(*
ExecuteSkill.Parameter[4].ID := ;
ExecuteSkill.Parameter[4].Name := '';
ExecuteSkill.Parameter[4].Value := ;
*)

(*
ExecuteSkill.Parameter[5].ID := ;
ExecuteSkill.Parameter[5].Name := '';
ExecuteSkill.Parameter[5].Value := ;
*)



ExecuteSkill();

StepDone := ExecuteSkill.Done;
END_ACTION

ACTION ST40_TransOutput_active:
//RT: 2014.11.23: Mover zum Output
StepDone := FALSE;

//Skill auswählen
ExecuteSkill.SkillID 		:= 1320;
ExecuteSkill.SkillName	 	:= 'Transport';

//Parameter setzen

ExecuteSkill.Parameter[3].ID := 3;
ExecuteSkill.Parameter[3].Name := 'Velocity';
ExecuteSkill.Parameter[3].Value := 300;



ExecuteSkill.Parameter[1].ID :=  1;
ExecuteSkill.Parameter[1].Name := 'TargetPosition X';
ExecuteSkill.Parameter[1].Value := 30 ;
ExecuteSkill.Parameter[1].StringValue := '#DP#2#XPosition';



ExecuteSkill.Parameter[2].ID := 2;
ExecuteSkill.Parameter[2].Name := 'TargetPosition Z';
ExecuteSkill.Parameter[2].Value := ZInputOutput;// ZCookieModule - ZCookieModuleCalibration - 2* Cookiethickness + toppingthickness+ Preasureheight  ;



(* ExecuteSkill.Parameter[4].ID := 4;
ExecuteSkill.Parameter[4].Name := 'Acceleration';
ExecuteSkill.Parameter[4].Value :=0 ;

*)
(*
ExecuteSkill.Parameter[5].ID := ;
ExecuteSkill.Parameter[5].Name := '';
ExecuteSkill.Parameter[5].Value := ;
*)



ExecuteSkill();

StepDone := ExecuteSkill.Done;
END_ACTION

ACTION ST43_UnblockOutput_active:
//RT: 2014.11.23: Gibt Mover Position Frei
StepDone := FALSE;

//Skill auswählen
ExecuteSkill.SkillID 		:= 1316;
ExecuteSkill.SkillName	 	:= 'Unblock';

//Parameter setzen

ExecuteSkill.Parameter[1].ID := 1;
ExecuteSkill.Parameter[1].Name := 'TaskID';
ExecuteSkill.Parameter[1].Value := Order.TaskID;


(*
ExecuteSkill.Parameter[2].ID := ;
ExecuteSkill.Parameter[2].Name := '';
ExecuteSkill.Parameter[2].Value := ;
*)

(*
ExecuteSkill.Parameter[3].ID := ;
ExecuteSkill.Parameter[3].Name := '';
ExecuteSkill.Parameter[3].Value := ;
*)

(*
ExecuteSkill.Parameter[4].ID := ;
ExecuteSkill.Parameter[4].Name := '';
ExecuteSkill.Parameter[4].Value := ;
*)

(*
ExecuteSkill.Parameter[5].ID := ;
ExecuteSkill.Parameter[5].Name := '';
ExecuteSkill.Parameter[5].Value := ;
*)



ExecuteSkill();

StepDone := ExecuteSkill.Done;
END_ACTION

ACTION ST4_Output_entry:
SectionReady := FALSE;
END_ACTION

ACTION ST3_Pump_active:
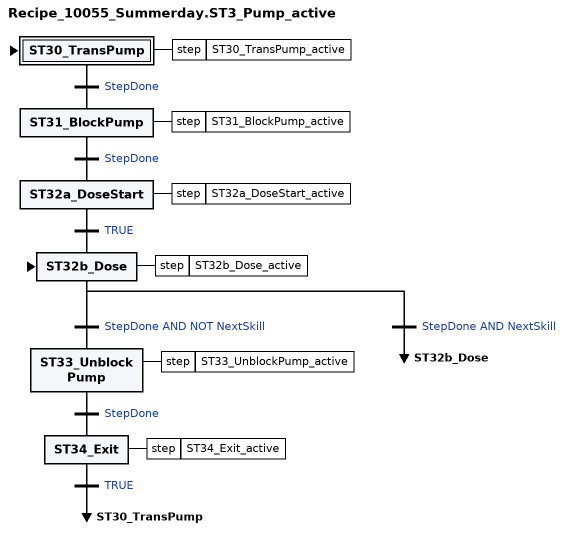
INITIAL_STEP ST30_TransPump:
    ST30_TransPump_active(N);  // step action
END_STEP
TRANSITION FROM ST30_TransPump TO ST31_BlockPump
    := StepDone;
END_TRANSITION
STEP ST31_BlockPump:
    ST31_BlockPump_active(N);  // step action
END_STEP
TRANSITION FROM ST31_BlockPump TO ST32a_DoseStart
    := StepDone;
END_TRANSITION
STEP ST32a_DoseStart:
    ST32a_DoseStart_active(N);  // step action
END_STEP
TRANSITION FROM ST32a_DoseStart TO ST32b_Dose
    := TRUE;
END_TRANSITION
STEP ST32b_Dose:
    ST32b_Dose_active(N);  // step action
END_STEP
TRANSITION FROM ST32b_Dose TO ST33_UnblockPump
    := StepDone AND NOT NextSkill;
END_TRANSITION
STEP ST33_UnblockPump:
    ST33_UnblockPump_active(N);  // step action
END_STEP
TRANSITION FROM ST33_UnblockPump TO ST34_Exit
    := StepDone;
END_TRANSITION
STEP ST34_Exit:
    ST34_Exit_active(N);  // step action
END_STEP
TRANSITION FROM ST34_Exit TO ST30_TransPump
    := TRUE;
END_TRANSITION
TRANSITION FROM ST32b_Dose TO ST32b_Dose
    := StepDone AND NextSkill;
END_TRANSITION
END_ACTION

ACTION ST41_BlockOutput_active:
//RT: 2014.11.23: Blockirt den Mover an Position
StepDone := FALSE;

//Skill auswählen
ExecuteSkill.SkillID 		:= 1315;
ExecuteSkill.SkillName	 	:= 'Block';

//Parameter setzen

ExecuteSkill.Parameter[1].ID := 1;
ExecuteSkill.Parameter[1].Name := 'TaskID';
ExecuteSkill.Parameter[1].Value := Order.TaskID;


(*
ExecuteSkill.Parameter[2].ID := ;
ExecuteSkill.Parameter[2].Name := '';
ExecuteSkill.Parameter[2].Value := ;
*)

(*
ExecuteSkill.Parameter[3].ID := ;
ExecuteSkill.Parameter[3].Name := '';
ExecuteSkill.Parameter[3].Value := ;
*)

(*
ExecuteSkill.Parameter[4].ID := ;
ExecuteSkill.Parameter[4].Name := '';
ExecuteSkill.Parameter[4].Value := ;
*)

(*
ExecuteSkill.Parameter[5].ID := ;
ExecuteSkill.Parameter[5].Name := '';
ExecuteSkill.Parameter[5].Value := ;
*)



ExecuteSkill();

StepDone := ExecuteSkill.Done;
END_ACTION

END_FUNCTION_BLOCK

// ---- POUs/Recipes/Recipe_10056_ArcturianSunrise.TcPOU
FUNCTION_BLOCK Recipe_10056_ArcturianSunrise
VAR_INPUT
	execute: BOOL;
	Order: DUT_RECIPEORDER;
END_VAR
VAR_OUTPUT
	RecipeInfo: DUT_RECIPEOFFER;
	RecipeDone: BOOL;
	InitDone: BOOL;
	Ready: BOOL;
END_VAR
VAR
	userparametersum: LREAL;
	StepDone: BOOL;
	i: INT;
	Command: ARRAY[1..5] OF DUT_RecipeCommand;
	NextSkill: BOOL;
	SectionReady: BOOL;
END_VAR

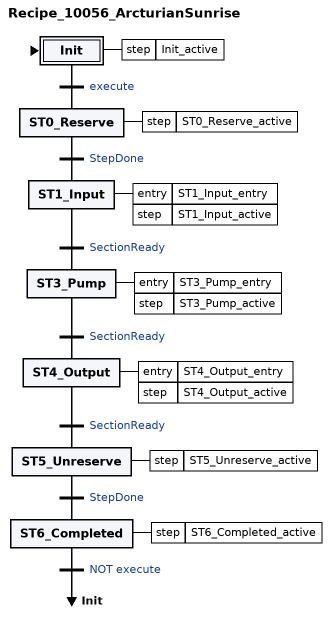
INITIAL_STEP Init:
    Init_active(N);  // step action
END_STEP
TRANSITION FROM Init TO ST0_Reserve
    := execute;
END_TRANSITION
STEP ST0_Reserve:
    ST0_Reserve_active(N);  // step action
END_STEP
TRANSITION FROM ST0_Reserve TO ST1_Input
    := StepDone;
END_TRANSITION
STEP ST1_Input:
    ST1_Input_entry(P1);  // entry action
    ST1_Input_active(N);  // step action
END_STEP
TRANSITION FROM ST1_Input TO ST3_Pump
    := SectionReady;
END_TRANSITION
STEP ST3_Pump:
    ST3_Pump_entry(P1);  // entry action
    ST3_Pump_active(N);  // step action
END_STEP
TRANSITION FROM ST3_Pump TO ST4_Output
    := SectionReady;
END_TRANSITION
STEP ST4_Output:
    ST4_Output_entry(P1);  // entry action
    ST4_Output_active(N);  // step action
END_STEP
TRANSITION FROM ST4_Output TO ST5_Unreserve
    := SectionReady;
END_TRANSITION
STEP ST5_Unreserve:
    ST5_Unreserve_active(N);  // step action
END_STEP
TRANSITION FROM ST5_Unreserve TO ST6_Completed
    := StepDone;
END_TRANSITION
STEP ST6_Completed:
    ST6_Completed_active(N);  // step action
END_STEP
TRANSITION FROM ST6_Completed TO Init
    := NOT execute;
END_TRANSITION

ACTION ST43_UnblockOutput_active:
//RT: 2014.11.23: Gibt Mover Position Frei
StepDone := FALSE;

//Skill auswählen
ExecuteSkill.SkillID 		:= 1316;
ExecuteSkill.SkillName	 	:= 'Unblock';

//Parameter setzen

ExecuteSkill.Parameter[1].ID := 1;
ExecuteSkill.Parameter[1].Name := 'TaskID';
ExecuteSkill.Parameter[1].Value := Order.TaskID;


(*
ExecuteSkill.Parameter[2].ID := ;
ExecuteSkill.Parameter[2].Name := '';
ExecuteSkill.Parameter[2].Value := ;
*)

(*
ExecuteSkill.Parameter[3].ID := ;
ExecuteSkill.Parameter[3].Name := '';
ExecuteSkill.Parameter[3].Value := ;
*)

(*
ExecuteSkill.Parameter[4].ID := ;
ExecuteSkill.Parameter[4].Name := '';
ExecuteSkill.Parameter[4].Value := ;
*)

(*
ExecuteSkill.Parameter[5].ID := ;
ExecuteSkill.Parameter[5].Name := '';
ExecuteSkill.Parameter[5].Value := ;
*)



ExecuteSkill();

StepDone := ExecuteSkill.Done;
END_ACTION

ACTION ST31_BlockPump_active:
//RT: 2014.11.23: Blockirt den Mover an Position
StepDone := FALSE;

//Skill auswählen
ExecuteSkill.SkillID 		:= 1315;
ExecuteSkill.SkillName	 	:= 'Block';

//Parameter setzen

ExecuteSkill.Parameter[1].ID := 1;
ExecuteSkill.Parameter[1].Name := 'TaskID';
ExecuteSkill.Parameter[1].Value := Order.TaskID;


(*
ExecuteSkill.Parameter[2].ID := ;
ExecuteSkill.Parameter[2].Name := '';
ExecuteSkill.Parameter[2].Value := ;
*)

(*
ExecuteSkill.Parameter[3].ID := ;
ExecuteSkill.Parameter[3].Name := '';
ExecuteSkill.Parameter[3].Value := ;
*)

(*
ExecuteSkill.Parameter[4].ID := ;
ExecuteSkill.Parameter[4].Name := '';
ExecuteSkill.Parameter[4].Value := ;
*)

(*
ExecuteSkill.Parameter[5].ID := ;
ExecuteSkill.Parameter[5].Name := '';
ExecuteSkill.Parameter[5].Value := ;
*)



ExecuteSkill();

StepDone := ExecuteSkill.Done;
END_ACTION

ACTION ST3_Pump_active:
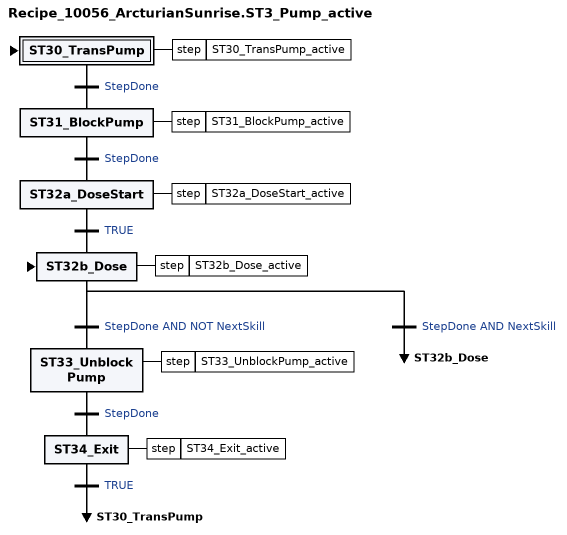
INITIAL_STEP ST30_TransPump:
    ST30_TransPump_active(N);  // step action
END_STEP
TRANSITION FROM ST30_TransPump TO ST31_BlockPump
    := StepDone;
END_TRANSITION
STEP ST31_BlockPump:
    ST31_BlockPump_active(N);  // step action
END_STEP
TRANSITION FROM ST31_BlockPump TO ST32a_DoseStart
    := StepDone;
END_TRANSITION
STEP ST32a_DoseStart:
    ST32a_DoseStart_active(N);  // step action
END_STEP
TRANSITION FROM ST32a_DoseStart TO ST32b_Dose
    := TRUE;
END_TRANSITION
STEP ST32b_Dose:
    ST32b_Dose_active(N);  // step action
END_STEP
TRANSITION FROM ST32b_Dose TO ST33_UnblockPump
    := StepDone AND NOT NextSkill;
END_TRANSITION
STEP ST33_UnblockPump:
    ST33_UnblockPump_active(N);  // step action
END_STEP
TRANSITION FROM ST33_UnblockPump TO ST34_Exit
    := StepDone;
END_TRANSITION
STEP ST34_Exit:
    ST34_Exit_active(N);  // step action
END_STEP
TRANSITION FROM ST34_Exit TO ST30_TransPump
    := TRUE;
END_TRANSITION
TRANSITION FROM ST32b_Dose TO ST32b_Dose
    := StepDone AND NextSkill;
END_TRANSITION
END_ACTION

ACTION ST44_Exit_active:
SectionReady := TRUE;
END_ACTION

ACTION ST13_UnblockInput_active:
//RT: 2014.11.23: Gibt Mover Position Frei
StepDone := FALSE;

//Skill auswählen
ExecuteSkill.SkillID 		:= 1316;
ExecuteSkill.SkillName	 	:= 'Unblock';

//Parameter setzen

ExecuteSkill.Parameter[1].ID := 1;
ExecuteSkill.Parameter[1].Name := 'TaskID';
ExecuteSkill.Parameter[1].Value := Order.TaskID;


(*
ExecuteSkill.Parameter[2].ID := ;
ExecuteSkill.Parameter[2].Name := '';
ExecuteSkill.Parameter[2].Value := ;
*)

(*
ExecuteSkill.Parameter[3].ID := ;
ExecuteSkill.Parameter[3].Name := '';
ExecuteSkill.Parameter[3].Value := ;
*)

(*
ExecuteSkill.Parameter[4].ID := ;
ExecuteSkill.Parameter[4].Name := '';
ExecuteSkill.Parameter[4].Value := ;
*)

(*
ExecuteSkill.Parameter[5].ID := ;
ExecuteSkill.Parameter[5].Name := '';
ExecuteSkill.Parameter[5].Value := ;
*)



ExecuteSkill();

StepDone := ExecuteSkill.Done;
END_ACTION

ACTION ST1_Input_active:
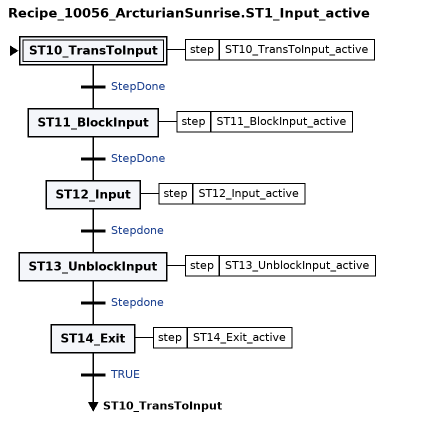
INITIAL_STEP ST10_TransToInput:
    ST10_TransToInput_active(N);  // step action
END_STEP
TRANSITION FROM ST10_TransToInput TO ST11_BlockInput
    := StepDone;
END_TRANSITION
STEP ST11_BlockInput:
    ST11_BlockInput_active(N);  // step action
END_STEP
TRANSITION FROM ST11_BlockInput TO ST12_Input
    := StepDone;
END_TRANSITION
STEP ST12_Input:
    ST12_Input_active(N);  // step action
END_STEP
TRANSITION FROM ST12_Input TO ST13_UnblockInput
    := Stepdone;
END_TRANSITION
STEP ST13_UnblockInput:
    ST13_UnblockInput_active(N);  // step action
END_STEP
TRANSITION FROM ST13_UnblockInput TO ST14_Exit
    := Stepdone;
END_TRANSITION
STEP ST14_Exit:
    ST14_Exit_active(N);  // step action
END_STEP
TRANSITION FROM ST14_Exit TO ST10_TransToInput
    := TRUE;
END_TRANSITION
END_ACTION

ACTION ST6_Completed_active:
//RT: 2014.11.23: Warte auf Execute = False
RecipeDone := TRUE;
StepDone := FALSE;
END_ACTION

ACTION ST32a_DoseStart_active:
//RT: 2014.11.23: Summe aller zutaten zum Normiren

userparametersum := 0;
FOR i := 1 TO UserParameterCnt DO
	IF NOT (order.UserParameter[i].Value = 0) THEN
		userparametersum := userparametersum + order.UserParameter[i].Value;
	
	END_IF
END_FOR
IF userparametersum = 0 THEN
userparametersum := -1;
END_IF

//RT: 2014.11.23: Start wert des Arrays setzen
i := 1;
NextSkill := TRUE ;
END_ACTION

ACTION ST11_BlockInput_active:
//RT: 2014.11.23: Blockirt den Mover an Position
StepDone := FALSE;

//Skill auswählen
ExecuteSkill.SkillID 		:= 1315;
ExecuteSkill.SkillName	 	:= 'Block';

//Parameter setzen

ExecuteSkill.Parameter[1].ID := 1;
ExecuteSkill.Parameter[1].Name := 'TaskID';
ExecuteSkill.Parameter[1].Value := Order.TaskID;


(*
ExecuteSkill.Parameter[2].ID := ;
ExecuteSkill.Parameter[2].Name := '';
ExecuteSkill.Parameter[2].Value := ;
*)

(*
ExecuteSkill.Parameter[3].ID := ;
ExecuteSkill.Parameter[3].Name := '';
ExecuteSkill.Parameter[3].Value := ;
*)

(*
ExecuteSkill.Parameter[4].ID := ;
ExecuteSkill.Parameter[4].Name := '';
ExecuteSkill.Parameter[4].Value := ;
*)

(*
ExecuteSkill.Parameter[5].ID := ;
ExecuteSkill.Parameter[5].Name := '';
ExecuteSkill.Parameter[5].Value := ;
*)



ExecuteSkill();

StepDone := ExecuteSkill.Done;
END_ACTION

ACTION ST5_Unreserve_active:
//RT: 2014.11.23: Mover Freigeben
StepDone := FALSE;

//Skill auswählen
ExecuteSkill.SkillID 		:= 1311;
ExecuteSkill.SkillName	 	:= 'Unreserve';

//Parameter setzen

ExecuteSkill.Parameter[1].ID := 1;
ExecuteSkill.Parameter[1].Name := 'TaskID';
ExecuteSkill.Parameter[1].Value := Order.TaskID;


(*
ExecuteSkill.Parameter[2].ID := ;
ExecuteSkill.Parameter[2].Name := '';
ExecuteSkill.Parameter[2].Val ue := ;
*)

(*
ExecuteSkill.Parameter[3].ID := ;
ExecuteSkill.Parameter[3].Name := '';
ExecuteSkill.Parameter[3].Value := ;
*)

(*
ExecuteSkill.Parameter[4].ID := ;
ExecuteSkill.Parameter[4].Name := '';
ExecuteSkill.Parameter[4].Value := ;
*)

(*
ExecuteSkill.Parameter[5].ID := ;
ExecuteSkill.Parameter[5].Name := '';
ExecuteSkill.Parameter[5].Value := ;
*)



ExecuteSkill();

StepDone := ExecuteSkill.Done;
END_ACTION

ACTION ST14_Exit_active:
SectionReady := TRUE;
END_ACTION

ACTION ST1_Reserve0_active:
//RT: 2014.11.23: Reservire einen Mover

StepDone := FALSE;
RecipeDone := FALSE;
//Skill auswählen
ExecuteSkill.SkillID 		:= 1310;
ExecuteSkill.SkillName	 	:= 'Reserve';

//Parameter setzen

ExecuteSkill.Parameter[1].ID := 1;
ExecuteSkill.Parameter[1].Name := 'TaskID';
ExecuteSkill.Parameter[1].Value := Order.TaskID;

(*
ExecuteSkill.Parameter[2].ID := ;
ExecuteSkill.Parameter[2].Name := '';
ExecuteSkill.Parameter[2].Value := ;
*)

(*
ExecuteSkill.Parameter[3].ID := ;
ExecuteSkill.Parameter[3].Name := '';
ExecuteSkill.Parameter[3].Value := ;
*)

(*
ExecuteSkill.Parameter[4].ID := ;
ExecuteSkill.Parameter[4].Name := '';
ExecuteSkill.Parameter[4].Value := ;
*)

(*
ExecuteSkill.Parameter[5].ID := ;
ExecuteSkill.Parameter[5].Name := '';
ExecuteSkill.Parameter[5].Value := ;
*)

ExecuteSkill();

StepDone := ExecuteSkill.Done;
END_ACTION

ACTION ST32b_Dose_active:
//RT: 2014.11.23: Die Dosir Skills anlegen
StepDone := FALSE;

//Skill auswählen
ExecuteSkill.SkillID 		:= Command[i].SkillID;
ExecuteSkill.SkillName	 	:= Command[i].SkillName;
//Parameter setzen

ExecuteSkill.Parameter[0].ID := 1;
ExecuteSkill.Parameter[0].Name := 'Quantity';
//order.userParameter[0] = amount
ExecuteSkill.Parameter[0].Value := order.UserParameter[0].Value * order.UserParameter[i].Value / userparametersum ;//Summe aller Zutatenmengen;

(*
ExecuteSkill.Parameter[2].ID := ;
ExecuteSkill.Parameter[2].Name := '';
ExecuteSkill.Parameter[2].Value := ;
*)

(*
ExecuteSkill.Parameter[3].ID := ;
ExecuteSkill.Parameter[3].Name := '';
ExecuteSkill.Parameter[3].Value := ;
*)

(*
ExecuteSkill.Parameter[4].ID := ;
ExecuteSkill.Parameter[4].Name := '';
ExecuteSkill.Parameter[4].Value := ;
*)

(*
ExecuteSkill.Parameter[5].ID := ;
ExecuteSkill.Parameter[5].Name := '';
ExecuteSkill.Parameter[5].Value := ;
*)


ExecuteSkill();

StepDone := ExecuteSkill.Done;

i := i + 1 ;

IF i = 6 THEN
	NextSkill := FALSE;
ELSIF Command[i].SkillID = 0 THEN
	NextSkill := FALSE;
ELSE
	NextSkill := TRUE;
END_IF
END_ACTION

ACTION ST3_Pump_entry:
SectionReady := FALSE;
END_ACTION

ACTION Init_active:
//RT: 2014.11.23: Vorbereiten der daten und der HMI
RecipeDone := FALSE;

// Initialisation of Recipe Parameters an name etc
RecipeInfo.Name := 'Blue Sunrise';
RecipeInfo.Description := 'Contrastful arrangement of sweet syrup and sour juice';
RecipeInfo.Dummy := FALSE;
RecipeInfo.RecipeID := 10056; 	// 
Initdone := TRUE;

//RT: 2014.11.23: wenn weniger als 5 alle lehren skills SkillID := 0
Command[1].SkillID := 1112;
Command[1].SkillName := 'Lemon Juice';
Command[1].Quantity := 30;

Command[2].SkillID := 1118;
Command[2].SkillName := 'Strawberry Syrup';
Command[2].Quantity := 8;

Command[3].SkillID := 1114;
Command[3].SkillName := 'Pineapple Juice';
Command[3].Quantity := 54;

Command[4].SkillID := 1111;
Command[4].SkillName := 'Blue Curacao';
Command[4].Quantity := 8;

Command[5].SkillID := 0;
Command[5].SkillName := 'Nothing';
Command[5].Quantity := 0;








//Parameter 0:

	RecipeInfo.UserParameter[0].Dummy 		:= FALSE;
	RecipeInfo.UserParameter[0].Default		:= 200;
	RecipeInfo.UserParameter[0].Description	:= 'Gives the total fluid amount in the glass';
	RecipeInfo.UserParameter[0].MaxValue	:= 200;
	RecipeInfo.UserParameter[0].MinValue	:= 10;
	RecipeInfo.UserParameter[0].Name		:= 'Total Liquid Amount';
	RecipeInfo.UserParameter[0].Unit		:= 'ml';
	
//Parameter 1-5:
FOR i := 1 TO 5 DO
	IF Command[i].SkillID = 0 THEN
		RecipeInfo.UserParameter[i].Dummy 		:= TRUE;
	ELSE
		RecipeInfo.UserParameter[i].Dummy 		:= FALSE;
		RecipeInfo.UserParameter[i].Default		:= Command[i].Quantity;
		RecipeInfo.UserParameter[i].Description	:= Command[i].SkillName;
		RecipeInfo.UserParameter[i].MaxValue	:= 100;
		RecipeInfo.UserParameter[i].MinValue	:= 1;
		RecipeInfo.UserParameter[i].Name		:= Command[i].SkillName;
		RecipeInfo.UserParameter[i].Unit		:= 'ml';	
	END_IF
END_FOR
END_ACTION

ACTION ST32b_Dose_exit:

END_ACTION

ACTION ST40_TransOutput_active:
//RT: 2014.11.23: Mover zum Output
StepDone := FALSE;

//Skill auswählen
ExecuteSkill.SkillID 		:= 1320;
ExecuteSkill.SkillName	 	:= 'Transport';

//Parameter setzen

ExecuteSkill.Parameter[3].ID := 3;
ExecuteSkill.Parameter[3].Name := 'Velocity';
ExecuteSkill.Parameter[3].Value := 300;



ExecuteSkill.Parameter[1].ID :=  1;
ExecuteSkill.Parameter[1].Name := 'TargetPosition X';
ExecuteSkill.Parameter[1].Value := 30 ;
ExecuteSkill.Parameter[1].StringValue := '#DP#2#XPosition';



ExecuteSkill.Parameter[2].ID := 2;
ExecuteSkill.Parameter[2].Name := 'TargetPosition Z';
ExecuteSkill.Parameter[2].Value := 100;// ZCookieModule - ZCookieModuleCalibration - 2* Cookiethickness + toppingthickness+ Preasureheight  ;



(* ExecuteSkill.Parameter[4].ID := 4;
ExecuteSkill.Parameter[4].Name := 'Acceleration';
ExecuteSkill.Parameter[4].Value :=0 ;

*)
(*
ExecuteSkill.Parameter[5].ID := ;
ExecuteSkill.Parameter[5].Name := '';
ExecuteSkill.Parameter[5].Value := ;
*)



ExecuteSkill();

StepDone := ExecuteSkill.Done;
END_ACTION

ACTION ST33_UnblockPump_active:
//RT: 2014.11.23: Gibt Mover Position Frei
StepDone := FALSE;

//Skill auswählen
ExecuteSkill.SkillID 		:= 1316;
ExecuteSkill.SkillName	 	:= 'Unblock';

//Parameter setzen

ExecuteSkill.Parameter[1].ID := 1;
ExecuteSkill.Parameter[1].Name := 'TaskID';
ExecuteSkill.Parameter[1].Value := Order.TaskID;


(*
ExecuteSkill.Parameter[2].ID := ;
ExecuteSkill.Parameter[2].Name := '';
ExecuteSkill.Parameter[2].Value := ;
*)

(*
ExecuteSkill.Parameter[3].ID := ;
ExecuteSkill.Parameter[3].Name := '';
ExecuteSkill.Parameter[3].Value := ;
*)

(*
ExecuteSkill.Parameter[4].ID := ;
ExecuteSkill.Parameter[4].Name := '';
ExecuteSkill.Parameter[4].Value := ;
*)

(*
ExecuteSkill.Parameter[5].ID := ;
ExecuteSkill.Parameter[5].Name := '';
ExecuteSkill.Parameter[5].Value := ;
*)



ExecuteSkill();

StepDone := ExecuteSkill.Done;
END_ACTION

ACTION ST0_Reserve_active:
//RT: 2014.11.23: Reservire einen Mover

StepDone := FALSE;
RecipeDone := FALSE;
//Skill auswählen
ExecuteSkill.SkillID 		:= 1310;
ExecuteSkill.SkillName	 	:= 'Reserve';

//Parameter setzen

ExecuteSkill.Parameter[1].ID := 1;
ExecuteSkill.Parameter[1].Name := 'TaskID';
ExecuteSkill.Parameter[1].Value := Order.TaskID;

(*
ExecuteSkill.Parameter[2].ID := ;
ExecuteSkill.Parameter[2].Name := '';
ExecuteSkill.Parameter[2].Value := ;
*)

(*
ExecuteSkill.Parameter[3].ID := ;
ExecuteSkill.Parameter[3].Name := '';
ExecuteSkill.Parameter[3].Value := ;
*)

(*
ExecuteSkill.Parameter[4].ID := ;
ExecuteSkill.Parameter[4].Name := '';
ExecuteSkill.Parameter[4].Value := ;
*)

(*
ExecuteSkill.Parameter[5].ID := ;
ExecuteSkill.Parameter[5].Name := '';
ExecuteSkill.Parameter[5].Value := ;
*)

ExecuteSkill();

StepDone := ExecuteSkill.Done;
END_ACTION

ACTION ST42_CocktailOutput_active:
//RT: 2014.11.23: Ausgeben des Produktes
StepDone := FALSE;

//Skill auswählen
ExecuteSkill.SkillID 		:= 1403;
ExecuteSkill.SkillName	 	:= 'Output';

//Parameter setzen

ExecuteSkill.Parameter[1].ID := 1;
ExecuteSkill.Parameter[1].Name := 'TaskID';
ExecuteSkill.Parameter[1].Value := Order.TaskID;


(*
ExecuteSkill.Parameter[2].ID := ;
ExecuteSkill.Parameter[2].Name := '';
ExecuteSkill.Parameter[2].Value := ;
*)

(*
ExecuteSkill.Parameter[3].ID := ;
ExecuteSkill.Parameter[3].Name := '';
ExecuteSkill.Parameter[3].Value := ;
*)

(*
ExecuteSkill.Parameter[4].ID := ;
ExecuteSkill.Parameter[4].Name := '';
ExecuteSkill.Parameter[4].Value := ;
*)

(*
ExecuteSkill.Parameter[5].ID := ;
ExecuteSkill.Parameter[5].Name := '';
ExecuteSkill.Parameter[5].Value := ;
*)



ExecuteSkill();

StepDone := ExecuteSkill.Done;
END_ACTION

ACTION ST4_Output_entry:
SectionReady := FALSE;
END_ACTION

ACTION ST4_Output_active:
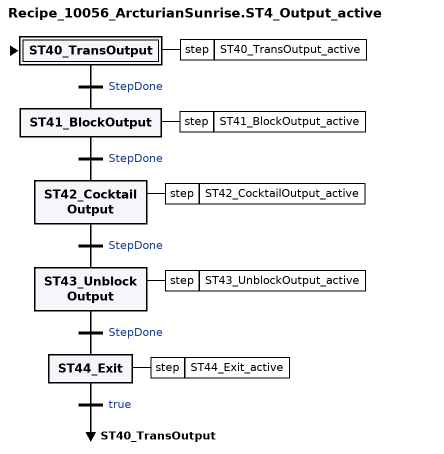
INITIAL_STEP ST40_TransOutput:
    ST40_TransOutput_active(N);  // step action
END_STEP
TRANSITION FROM ST40_TransOutput TO ST41_BlockOutput
    := StepDone;
END_TRANSITION
STEP ST41_BlockOutput:
    ST41_BlockOutput_active(N);  // step action
END_STEP
TRANSITION FROM ST41_BlockOutput TO ST42_CocktailOutput
    := StepDone;
END_TRANSITION
STEP ST42_CocktailOutput:
    ST42_CocktailOutput_active(N);  // step action
END_STEP
TRANSITION FROM ST42_CocktailOutput TO ST43_UnblockOutput
    := StepDone;
END_TRANSITION
STEP ST43_UnblockOutput:
    ST43_UnblockOutput_active(N);  // step action
END_STEP
TRANSITION FROM ST43_UnblockOutput TO ST44_Exit
    := StepDone;
END_TRANSITION
STEP ST44_Exit:
    ST44_Exit_active(N);  // step action
END_STEP
TRANSITION FROM ST44_Exit TO ST40_TransOutput
    := true;
END_TRANSITION
END_ACTION

ACTION ST30_TransPump_active:
//RT: 2014.11.23: Mover zum Pump
StepDone := FALSE;

//Skill auswählen
ExecuteSkill.SkillID 		:= 1320;
ExecuteSkill.SkillName	 	:= 'Transport';

//Parameter setzen

ExecuteSkill.Parameter[3].ID := 3;
ExecuteSkill.Parameter[3].Name := 'Velocity';
ExecuteSkill.Parameter[3].Value := 1000;



ExecuteSkill.Parameter[1].ID :=  1;
ExecuteSkill.Parameter[1].Name := 'TargetPosition X';
ExecuteSkill.Parameter[1].Value := 30 ;
ExecuteSkill.Parameter[1].StringValue := '#DP#2#XPosition';



ExecuteSkill.Parameter[2].ID := 2;
ExecuteSkill.Parameter[2].Name := 'TargetPosition Z';
ExecuteSkill.Parameter[2].Value := 25;// ZCookieModule - ZCookieModuleCalibration - 2* Cookiethickness + toppingthickness+ Preasureheight  ;



(*
ExecuteSkill.Parameter[4].ID := 4;
ExecuteSkill.Parameter[4].Name := 'Acceleration';
ExecuteSkill.Parameter[4].Value := 0 ;
*)

(*
ExecuteSkill.Parameter[5].ID := ;
ExecuteSkill.Parameter[5].Name := '';
ExecuteSkill.Parameter[5].Value := ;
*)



ExecuteSkill();

StepDone := ExecuteSkill.Done;
END_ACTION

ACTION ST10_TransToInput_active:
//RT: 2014.11.23: Mover zum Input

StepDone := FALSE;

//Skill auswählen
ExecuteSkill.SkillID 		:= 1320;
ExecuteSkill.SkillName	 	:= 'Transport';

//Parameter setzen

ExecuteSkill.Parameter[3].ID := 3;
ExecuteSkill.Parameter[3].Name := 'Velocity';
ExecuteSkill.Parameter[3].Value := 1000;



ExecuteSkill.Parameter[1].ID :=  1;
ExecuteSkill.Parameter[1].Name := 'TargetPosition X';
ExecuteSkill.Parameter[1].Value := 30 ;
ExecuteSkill.Parameter[1].StringValue := '#DP#2#XPosition';



ExecuteSkill.Parameter[2].ID := 2;
ExecuteSkill.Parameter[2].Name := 'TargetPosition Z';
ExecuteSkill.Parameter[2].Value := 100;// ZCookieModule - ZCookieModuleCalibration - 2* Cookiethickness + toppingthickness+ Preasureheight  ;



(*
ExecuteSkill.Parameter[4].ID := 4;
ExecuteSkill.Parameter[4].Name := 'Acceleration';
ExecuteSkill.Parameter[4].Value := 0 ;
*)

(*
ExecuteSkill.Parameter[5].ID := ;
ExecuteSkill.Parameter[5].Name := '';
ExecuteSkill.Parameter[5].Value := ;
*)



ExecuteSkill();

StepDone := ExecuteSkill.Done;
END_ACTION

ACTION ST12_Input_active:
//RT: 2014.11.23: Input Modul auslösen
StepDone := FALSE;

//Skill auswählen
ExecuteSkill.SkillID 		:= 1402;
ExecuteSkill.SkillName	 	:= 'Input';

//Parameter setzen

ExecuteSkill.Parameter[1].ID := 1;
ExecuteSkill.Parameter[1].Name := 'TaskID';
ExecuteSkill.Parameter[1].Value := Order.TaskID;


(*
ExecuteSkill.Parameter[2].ID := ;
ExecuteSkill.Parameter[2].Name := '';
ExecuteSkill.Parameter[2].Value := ;
*)

(*
ExecuteSkill.Parameter[3].ID := ;
ExecuteSkill.Parameter[3].Name := '';
ExecuteSkill.Parameter[3].Value := ;
*)

(*
ExecuteSkill.Parameter[4].ID := ;
ExecuteSkill.Parameter[4].Name := '';
ExecuteSkill.Parameter[4].Value := ;
*)

(*
ExecuteSkill.Parameter[5].ID := ;
ExecuteSkill.Parameter[5].Name := '';
ExecuteSkill.Parameter[5].Value := ;
*)



ExecuteSkill();

StepDone := ExecuteSkill.Done;
END_ACTION

ACTION ST41_BlockOutput_active:
//RT: 2014.11.23: Blockirt den Mover an Position
StepDone := FALSE;

//Skill auswählen
ExecuteSkill.SkillID 		:= 1315;
ExecuteSkill.SkillName	 	:= 'Block';

//Parameter setzen

ExecuteSkill.Parameter[1].ID := 1;
ExecuteSkill.Parameter[1].Name := 'TaskID';
ExecuteSkill.Parameter[1].Value := Order.TaskID;


(*
ExecuteSkill.Parameter[2].ID := ;
ExecuteSkill.Parameter[2].Name := '';
ExecuteSkill.Parameter[2].Value := ;
*)

(*
ExecuteSkill.Parameter[3].ID := ;
ExecuteSkill.Parameter[3].Name := '';
ExecuteSkill.Parameter[3].Value := ;
*)

(*
ExecuteSkill.Parameter[4].ID := ;
ExecuteSkill.Parameter[4].Name := '';
ExecuteSkill.Parameter[4].Value := ;
*)

(*
ExecuteSkill.Parameter[5].ID := ;
ExecuteSkill.Parameter[5].Name := '';
ExecuteSkill.Parameter[5].Value := ;
*)



ExecuteSkill();

StepDone := ExecuteSkill.Done;
END_ACTION

ACTION ST1_Input_entry:
SectionReady := FALSE;
END_ACTION

ACTION ST34_Exit_active:
SectionReady := TRUE;
END_ACTION

END_FUNCTION_BLOCK

// ---- POUs/Recipes/Recipe_10057_GreenFive.TcPOU
FUNCTION_BLOCK Recipe_10057_GreenFive
VAR_INPUT
	execute: BOOL;
	Order: DUT_RECIPEORDER;
END_VAR
VAR_OUTPUT
	RecipeInfo: DUT_RECIPEOFFER;
	RecipeDone: BOOL;
	InitDone: BOOL;
	Ready: BOOL;
END_VAR
VAR
	userparametersum: LREAL;
	StepDone: BOOL;
	i: INT;
	Command: ARRAY[1..5] OF DUT_RecipeCommand;
	NextSkill: BOOL;
	SectionReady: BOOL;
END_VAR

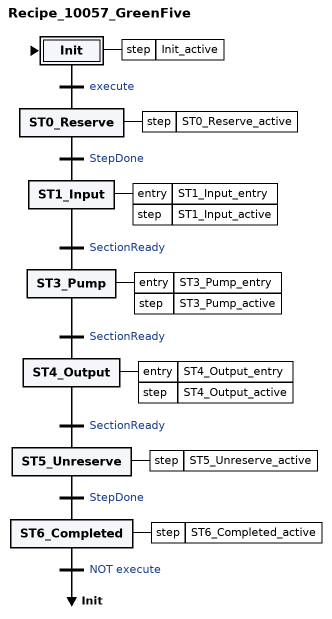
INITIAL_STEP Init:
    Init_active(N);  // step action
END_STEP
TRANSITION FROM Init TO ST0_Reserve
    := execute;
END_TRANSITION
STEP ST0_Reserve:
    ST0_Reserve_active(N);  // step action
END_STEP
TRANSITION FROM ST0_Reserve TO ST1_Input
    := StepDone;
END_TRANSITION
STEP ST1_Input:
    ST1_Input_entry(P1);  // entry action
    ST1_Input_active(N);  // step action
END_STEP
TRANSITION FROM ST1_Input TO ST3_Pump
    := SectionReady;
END_TRANSITION
STEP ST3_Pump:
    ST3_Pump_entry(P1);  // entry action
    ST3_Pump_active(N);  // step action
END_STEP
TRANSITION FROM ST3_Pump TO ST4_Output
    := SectionReady;
END_TRANSITION
STEP ST4_Output:
    ST4_Output_entry(P1);  // entry action
    ST4_Output_active(N);  // step action
END_STEP
TRANSITION FROM ST4_Output TO ST5_Unreserve
    := SectionReady;
END_TRANSITION
STEP ST5_Unreserve:
    ST5_Unreserve_active(N);  // step action
END_STEP
TRANSITION FROM ST5_Unreserve TO ST6_Completed
    := StepDone;
END_TRANSITION
STEP ST6_Completed:
    ST6_Completed_active(N);  // step action
END_STEP
TRANSITION FROM ST6_Completed TO Init
    := NOT execute;
END_TRANSITION

ACTION ST6_Completed_active:
//RT: 2014.11.23: Warte auf Execute = False
RecipeDone := TRUE;
StepDone := FALSE;
END_ACTION

ACTION ST1_Input_entry:
SectionReady := FALSE;
END_ACTION

ACTION ST3_Pump_entry:
SectionReady := FALSE;
END_ACTION

ACTION ST32b_Dose_active:
//RT: 2014.11.23: Die Dosir Skills anlegen
StepDone := FALSE;

//Skill auswählen
ExecuteSkill.SkillID 		:= Command[i].SkillID;
ExecuteSkill.SkillName	 	:= Command[i].SkillName;
//Parameter setzen

ExecuteSkill.Parameter[0].ID := 1;
ExecuteSkill.Parameter[0].Name := 'Quantity';
//order.userParameter[0] = amount
ExecuteSkill.Parameter[0].Value := order.UserParameter[0].Value * order.UserParameter[i].Value / userparametersum ;//Summe aller Zutatenmengen;

(*
ExecuteSkill.Parameter[2].ID := ;
ExecuteSkill.Parameter[2].Name := '';
ExecuteSkill.Parameter[2].Value := ;
*)

(*
ExecuteSkill.Parameter[3].ID := ;
ExecuteSkill.Parameter[3].Name := '';
ExecuteSkill.Parameter[3].Value := ;
*)

(*
ExecuteSkill.Parameter[4].ID := ;
ExecuteSkill.Parameter[4].Name := '';
ExecuteSkill.Parameter[4].Value := ;
*)

(*
ExecuteSkill.Parameter[5].ID := ;
ExecuteSkill.Parameter[5].Name := '';
ExecuteSkill.Parameter[5].Value := ;
*)


ExecuteSkill();

StepDone := ExecuteSkill.Done;

i := i + 1 ;

IF i = 6 THEN
	NextSkill := FALSE;
ELSIF Command[i].SkillID = 0 THEN
	NextSkill := FALSE;
ELSE
	NextSkill := TRUE;
END_IF
END_ACTION

ACTION ST32a_DoseStart_active:
//RT: 2014.11.23: Summe aller zutaten zum Normiren

userparametersum := 0;
FOR i := 1 TO UserParameterCnt DO
	IF NOT (order.UserParameter[i].Value = 0) THEN
		userparametersum := userparametersum + order.UserParameter[i].Value;
	
	END_IF
END_FOR
IF userparametersum = 0 THEN
userparametersum := -1;
END_IF

//RT: 2014.11.23: Start wert des Arrays setzen
i := 1;
NextSkill := TRUE ;
END_ACTION

ACTION ST12_Input_active:
//RT: 2014.11.23: Input Modul auslösen
StepDone := FALSE;

//Skill auswählen
ExecuteSkill.SkillID 		:= 1402;
ExecuteSkill.SkillName	 	:= 'Input';

//Parameter setzen

ExecuteSkill.Parameter[1].ID := 1;
ExecuteSkill.Parameter[1].Name := 'TaskID';
ExecuteSkill.Parameter[1].Value := Order.TaskID;


(*
ExecuteSkill.Parameter[2].ID := ;
ExecuteSkill.Parameter[2].Name := '';
ExecuteSkill.Parameter[2].Value := ;
*)

(*
ExecuteSkill.Parameter[3].ID := ;
ExecuteSkill.Parameter[3].Name := '';
ExecuteSkill.Parameter[3].Value := ;
*)

(*
ExecuteSkill.Parameter[4].ID := ;
ExecuteSkill.Parameter[4].Name := '';
ExecuteSkill.Parameter[4].Value := ;
*)

(*
ExecuteSkill.Parameter[5].ID := ;
ExecuteSkill.Parameter[5].Name := '';
ExecuteSkill.Parameter[5].Value := ;
*)



ExecuteSkill();

StepDone := ExecuteSkill.Done;
END_ACTION

ACTION ST3_Pump_active:
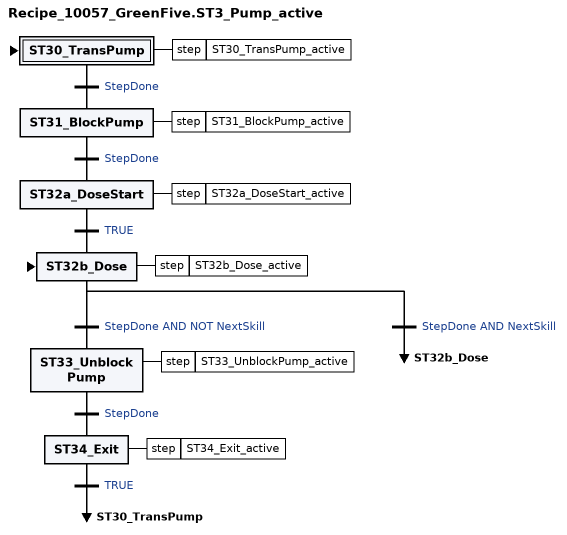
INITIAL_STEP ST30_TransPump:
    ST30_TransPump_active(N);  // step action
END_STEP
TRANSITION FROM ST30_TransPump TO ST31_BlockPump
    := StepDone;
END_TRANSITION
STEP ST31_BlockPump:
    ST31_BlockPump_active(N);  // step action
END_STEP
TRANSITION FROM ST31_BlockPump TO ST32a_DoseStart
    := StepDone;
END_TRANSITION
STEP ST32a_DoseStart:
    ST32a_DoseStart_active(N);  // step action
END_STEP
TRANSITION FROM ST32a_DoseStart TO ST32b_Dose
    := TRUE;
END_TRANSITION
STEP ST32b_Dose:
    ST32b_Dose_active(N);  // step action
END_STEP
TRANSITION FROM ST32b_Dose TO ST33_UnblockPump
    := StepDone AND NOT NextSkill;
END_TRANSITION
STEP ST33_UnblockPump:
    ST33_UnblockPump_active(N);  // step action
END_STEP
TRANSITION FROM ST33_UnblockPump TO ST34_Exit
    := StepDone;
END_TRANSITION
STEP ST34_Exit:
    ST34_Exit_active(N);  // step action
END_STEP
TRANSITION FROM ST34_Exit TO ST30_TransPump
    := TRUE;
END_TRANSITION
TRANSITION FROM ST32b_Dose TO ST32b_Dose
    := StepDone AND NextSkill;
END_TRANSITION
END_ACTION

ACTION ST34_Exit_active:
SectionReady := TRUE;
END_ACTION

ACTION ST32b_Dose_exit:

END_ACTION

ACTION ST44_Exit_active:
SectionReady := TRUE;
END_ACTION

ACTION ST10_TransToInput_active:
//RT: 2014.11.23: Mover zum Input

StepDone := FALSE;

//Skill auswählen
ExecuteSkill.SkillID 		:= 1320;
ExecuteSkill.SkillName	 	:= 'Transport';

//Parameter setzen

ExecuteSkill.Parameter[3].ID := 3;
ExecuteSkill.Parameter[3].Name := 'Velocity';
ExecuteSkill.Parameter[3].Value := 1000;



ExecuteSkill.Parameter[1].ID :=  1;
ExecuteSkill.Parameter[1].Name := 'TargetPosition X';
ExecuteSkill.Parameter[1].Value := 30 ;
ExecuteSkill.Parameter[1].StringValue := '#DP#2#XPosition';



ExecuteSkill.Parameter[2].ID := 2;
ExecuteSkill.Parameter[2].Name := 'TargetPosition Z';
ExecuteSkill.Parameter[2].Value := 100;// ZCookieModule - ZCookieModuleCalibration - 2* Cookiethickness + toppingthickness+ Preasureheight  ;



(*
ExecuteSkill.Parameter[4].ID := 4;
ExecuteSkill.Parameter[4].Name := 'Acceleration';
ExecuteSkill.Parameter[4].Value := 0 ;
*)

(*
ExecuteSkill.Parameter[5].ID := ;
ExecuteSkill.Parameter[5].Name := '';
ExecuteSkill.Parameter[5].Value := ;
*)



ExecuteSkill();

StepDone := ExecuteSkill.Done;
END_ACTION

ACTION ST4_Output_entry:
SectionReady := FALSE;
END_ACTION

ACTION ST42_CocktailOutput_active:
//RT: 2014.11.23: Ausgeben des Produktes
StepDone := FALSE;

//Skill auswählen
ExecuteSkill.SkillID 		:= 1403;
ExecuteSkill.SkillName	 	:= 'Output';

//Parameter setzen

ExecuteSkill.Parameter[1].ID := 1;
ExecuteSkill.Parameter[1].Name := 'TaskID';
ExecuteSkill.Parameter[1].Value := Order.TaskID;


(*
ExecuteSkill.Parameter[2].ID := ;
ExecuteSkill.Parameter[2].Name := '';
ExecuteSkill.Parameter[2].Value := ;
*)

(*
ExecuteSkill.Parameter[3].ID := ;
ExecuteSkill.Parameter[3].Name := '';
ExecuteSkill.Parameter[3].Value := ;
*)

(*
ExecuteSkill.Parameter[4].ID := ;
ExecuteSkill.Parameter[4].Name := '';
ExecuteSkill.Parameter[4].Value := ;
*)

(*
ExecuteSkill.Parameter[5].ID := ;
ExecuteSkill.Parameter[5].Name := '';
ExecuteSkill.Parameter[5].Value := ;
*)



ExecuteSkill();

StepDone := ExecuteSkill.Done;
END_ACTION

ACTION ST5_Unreserve_active:
//RT: 2014.11.23: Mover Freigeben
StepDone := FALSE;

//Skill auswählen
ExecuteSkill.SkillID 		:= 1311;
ExecuteSkill.SkillName	 	:= 'Unreserve';

//Parameter setzen

ExecuteSkill.Parameter[1].ID := 1;
ExecuteSkill.Parameter[1].Name := 'TaskID';
ExecuteSkill.Parameter[1].Value := Order.TaskID;


(*
ExecuteSkill.Parameter[2].ID := ;
ExecuteSkill.Parameter[2].Name := '';
ExecuteSkill.Parameter[2].Val ue := ;
*)

(*
ExecuteSkill.Parameter[3].ID := ;
ExecuteSkill.Parameter[3].Name := '';
ExecuteSkill.Parameter[3].Value := ;
*)

(*
ExecuteSkill.Parameter[4].ID := ;
ExecuteSkill.Parameter[4].Name := '';
ExecuteSkill.Parameter[4].Value := ;
*)

(*
ExecuteSkill.Parameter[5].ID := ;
ExecuteSkill.Parameter[5].Name := '';
ExecuteSkill.Parameter[5].Value := ;
*)



ExecuteSkill();

StepDone := ExecuteSkill.Done;
END_ACTION

ACTION ST11_BlockInput_active:
//RT: 2014.11.23: Blockirt den Mover an Position
StepDone := FALSE;

//Skill auswählen
ExecuteSkill.SkillID 		:= 1315;
ExecuteSkill.SkillName	 	:= 'Block';

//Parameter setzen

ExecuteSkill.Parameter[1].ID := 1;
ExecuteSkill.Parameter[1].Name := 'TaskID';
ExecuteSkill.Parameter[1].Value := Order.TaskID;


(*
ExecuteSkill.Parameter[2].ID := ;
ExecuteSkill.Parameter[2].Name := '';
ExecuteSkill.Parameter[2].Value := ;
*)

(*
ExecuteSkill.Parameter[3].ID := ;
ExecuteSkill.Parameter[3].Name := '';
ExecuteSkill.Parameter[3].Value := ;
*)

(*
ExecuteSkill.Parameter[4].ID := ;
ExecuteSkill.Parameter[4].Name := '';
ExecuteSkill.Parameter[4].Value := ;
*)

(*
ExecuteSkill.Parameter[5].ID := ;
ExecuteSkill.Parameter[5].Name := '';
ExecuteSkill.Parameter[5].Value := ;
*)



ExecuteSkill();

StepDone := ExecuteSkill.Done;
END_ACTION

ACTION ST13_UnblockInput_active:
//RT: 2014.11.23: Gibt Mover Position Frei
StepDone := FALSE;

//Skill auswählen
ExecuteSkill.SkillID 		:= 1316;
ExecuteSkill.SkillName	 	:= 'Unblock';

//Parameter setzen

ExecuteSkill.Parameter[1].ID := 1;
ExecuteSkill.Parameter[1].Name := 'TaskID';
ExecuteSkill.Parameter[1].Value := Order.TaskID;


(*
ExecuteSkill.Parameter[2].ID := ;
ExecuteSkill.Parameter[2].Name := '';
ExecuteSkill.Parameter[2].Value := ;
*)

(*
ExecuteSkill.Parameter[3].ID := ;
ExecuteSkill.Parameter[3].Name := '';
ExecuteSkill.Parameter[3].Value := ;
*)

(*
ExecuteSkill.Parameter[4].ID := ;
ExecuteSkill.Parameter[4].Name := '';
ExecuteSkill.Parameter[4].Value := ;
*)

(*
ExecuteSkill.Parameter[5].ID := ;
ExecuteSkill.Parameter[5].Name := '';
ExecuteSkill.Parameter[5].Value := ;
*)



ExecuteSkill();

StepDone := ExecuteSkill.Done;
END_ACTION

ACTION ST4_Output_active:
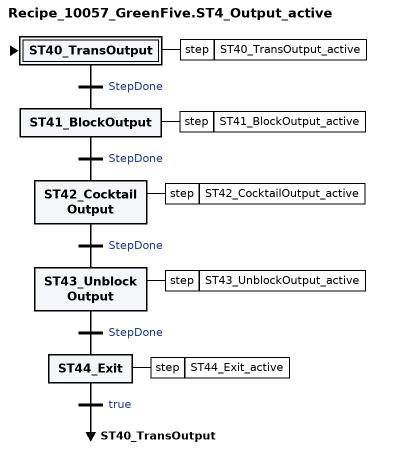
INITIAL_STEP ST40_TransOutput:
    ST40_TransOutput_active(N);  // step action
END_STEP
TRANSITION FROM ST40_TransOutput TO ST41_BlockOutput
    := StepDone;
END_TRANSITION
STEP ST41_BlockOutput:
    ST41_BlockOutput_active(N);  // step action
END_STEP
TRANSITION FROM ST41_BlockOutput TO ST42_CocktailOutput
    := StepDone;
END_TRANSITION
STEP ST42_CocktailOutput:
    ST42_CocktailOutput_active(N);  // step action
END_STEP
TRANSITION FROM ST42_CocktailOutput TO ST43_UnblockOutput
    := StepDone;
END_TRANSITION
STEP ST43_UnblockOutput:
    ST43_UnblockOutput_active(N);  // step action
END_STEP
TRANSITION FROM ST43_UnblockOutput TO ST44_Exit
    := StepDone;
END_TRANSITION
STEP ST44_Exit:
    ST44_Exit_active(N);  // step action
END_STEP
TRANSITION FROM ST44_Exit TO ST40_TransOutput
    := true;
END_TRANSITION
END_ACTION

ACTION ST0_Reserve_active:
//RT: 2014.11.23: Reservire einen Mover

StepDone := FALSE;
RecipeDone := FALSE;
//Skill auswählen
ExecuteSkill.SkillID 		:= 1310;
ExecuteSkill.SkillName	 	:= 'Reserve';

//Parameter setzen

ExecuteSkill.Parameter[1].ID := 1;
ExecuteSkill.Parameter[1].Name := 'TaskID';
ExecuteSkill.Parameter[1].Value := Order.TaskID;

(*
ExecuteSkill.Parameter[2].ID := ;
ExecuteSkill.Parameter[2].Name := '';
ExecuteSkill.Parameter[2].Value := ;
*)

(*
ExecuteSkill.Parameter[3].ID := ;
ExecuteSkill.Parameter[3].Name := '';
ExecuteSkill.Parameter[3].Value := ;
*)

(*
ExecuteSkill.Parameter[4].ID := ;
ExecuteSkill.Parameter[4].Name := '';
ExecuteSkill.Parameter[4].Value := ;
*)

(*
ExecuteSkill.Parameter[5].ID := ;
ExecuteSkill.Parameter[5].Name := '';
ExecuteSkill.Parameter[5].Value := ;
*)

ExecuteSkill();

StepDone := ExecuteSkill.Done;
END_ACTION

ACTION ST1_Reserve0_active:
//RT: 2014.11.23: Reservire einen Mover

StepDone := FALSE;
RecipeDone := FALSE;
//Skill auswählen
ExecuteSkill.SkillID 		:= 1310;
ExecuteSkill.SkillName	 	:= 'Reserve';

//Parameter setzen

ExecuteSkill.Parameter[1].ID := 1;
ExecuteSkill.Parameter[1].Name := 'TaskID';
ExecuteSkill.Parameter[1].Value := Order.TaskID;

(*
ExecuteSkill.Parameter[2].ID := ;
ExecuteSkill.Parameter[2].Name := '';
ExecuteSkill.Parameter[2].Value := ;
*)

(*
ExecuteSkill.Parameter[3].ID := ;
ExecuteSkill.Parameter[3].Name := '';
ExecuteSkill.Parameter[3].Value := ;
*)

(*
ExecuteSkill.Parameter[4].ID := ;
ExecuteSkill.Parameter[4].Name := '';
ExecuteSkill.Parameter[4].Value := ;
*)

(*
ExecuteSkill.Parameter[5].ID := ;
ExecuteSkill.Parameter[5].Name := '';
ExecuteSkill.Parameter[5].Value := ;
*)

ExecuteSkill();

StepDone := ExecuteSkill.Done;
END_ACTION

ACTION ST33_UnblockPump_active:
//RT: 2014.11.23: Gibt Mover Position Frei
StepDone := FALSE;

//Skill auswählen
ExecuteSkill.SkillID 		:= 1316;
ExecuteSkill.SkillName	 	:= 'Unblock';

//Parameter setzen

ExecuteSkill.Parameter[1].ID := 1;
ExecuteSkill.Parameter[1].Name := 'TaskID';
ExecuteSkill.Parameter[1].Value := Order.TaskID;


(*
ExecuteSkill.Parameter[2].ID := ;
ExecuteSkill.Parameter[2].Name := '';
ExecuteSkill.Parameter[2].Value := ;
*)

(*
ExecuteSkill.Parameter[3].ID := ;
ExecuteSkill.Parameter[3].Name := '';
ExecuteSkill.Parameter[3].Value := ;
*)

(*
ExecuteSkill.Parameter[4].ID := ;
ExecuteSkill.Parameter[4].Name := '';
ExecuteSkill.Parameter[4].Value := ;
*)

(*
ExecuteSkill.Parameter[5].ID := ;
ExecuteSkill.Parameter[5].Name := '';
ExecuteSkill.Parameter[5].Value := ;
*)



ExecuteSkill();

StepDone := ExecuteSkill.Done;
END_ACTION

ACTION ST43_UnblockOutput_active:
//RT: 2014.11.23: Gibt Mover Position Frei
StepDone := FALSE;

//Skill auswählen
ExecuteSkill.SkillID 		:= 1316;
ExecuteSkill.SkillName	 	:= 'Unblock';

//Parameter setzen

ExecuteSkill.Parameter[1].ID := 1;
ExecuteSkill.Parameter[1].Name := 'TaskID';
ExecuteSkill.Parameter[1].Value := Order.TaskID;


(*
ExecuteSkill.Parameter[2].ID := ;
ExecuteSkill.Parameter[2].Name := '';
ExecuteSkill.Parameter[2].Value := ;
*)

(*
ExecuteSkill.Parameter[3].ID := ;
ExecuteSkill.Parameter[3].Name := '';
ExecuteSkill.Parameter[3].Value := ;
*)

(*
ExecuteSkill.Parameter[4].ID := ;
ExecuteSkill.Parameter[4].Name := '';
ExecuteSkill.Parameter[4].Value := ;
*)

(*
ExecuteSkill.Parameter[5].ID := ;
ExecuteSkill.Parameter[5].Name := '';
ExecuteSkill.Parameter[5].Value := ;
*)



ExecuteSkill();

StepDone := ExecuteSkill.Done;
END_ACTION

ACTION ST14_Exit_active:
SectionReady := TRUE;
END_ACTION

ACTION ST41_BlockOutput_active:
//RT: 2014.11.23: Blockirt den Mover an Position
StepDone := FALSE;

//Skill auswählen
ExecuteSkill.SkillID 		:= 1315;
ExecuteSkill.SkillName	 	:= 'Block';

//Parameter setzen

ExecuteSkill.Parameter[1].ID := 1;
ExecuteSkill.Parameter[1].Name := 'TaskID';
ExecuteSkill.Parameter[1].Value := Order.TaskID;


(*
ExecuteSkill.Parameter[2].ID := ;
ExecuteSkill.Parameter[2].Name := '';
ExecuteSkill.Parameter[2].Value := ;
*)

(*
ExecuteSkill.Parameter[3].ID := ;
ExecuteSkill.Parameter[3].Name := '';
ExecuteSkill.Parameter[3].Value := ;
*)

(*
ExecuteSkill.Parameter[4].ID := ;
ExecuteSkill.Parameter[4].Name := '';
ExecuteSkill.Parameter[4].Value := ;
*)

(*
ExecuteSkill.Parameter[5].ID := ;
ExecuteSkill.Parameter[5].Name := '';
ExecuteSkill.Parameter[5].Value := ;
*)



ExecuteSkill();

StepDone := ExecuteSkill.Done;
END_ACTION

ACTION ST30_TransPump_active:
//RT: 2014.11.23: Mover zum Pump
StepDone := FALSE;

//Skill auswählen
ExecuteSkill.SkillID 		:= 1320;
ExecuteSkill.SkillName	 	:= 'Transport';

//Parameter setzen

ExecuteSkill.Parameter[3].ID := 3;
ExecuteSkill.Parameter[3].Name := 'Velocity';
ExecuteSkill.Parameter[3].Value := 1000;



ExecuteSkill.Parameter[1].ID :=  1;
ExecuteSkill.Parameter[1].Name := 'TargetPosition X';
ExecuteSkill.Parameter[1].Value := 30 ;
ExecuteSkill.Parameter[1].StringValue := '#DP#2#XPosition';



ExecuteSkill.Parameter[2].ID := 2;
ExecuteSkill.Parameter[2].Name := 'TargetPosition Z';
ExecuteSkill.Parameter[2].Value := 25;// ZCookieModule - ZCookieModuleCalibration - 2* Cookiethickness + toppingthickness+ Preasureheight  ;



(*
ExecuteSkill.Parameter[4].ID := 4;
ExecuteSkill.Parameter[4].Name := 'Acceleration';
ExecuteSkill.Parameter[4].Value := 0 ;
*)

(*
ExecuteSkill.Parameter[5].ID := ;
ExecuteSkill.Parameter[5].Name := '';
ExecuteSkill.Parameter[5].Value := ;
*)



ExecuteSkill();

StepDone := ExecuteSkill.Done;
END_ACTION

ACTION ST40_TransOutput_active:
//RT: 2014.11.23: Mover zum Output
StepDone := FALSE;

//Skill auswählen
ExecuteSkill.SkillID 		:= 1320;
ExecuteSkill.SkillName	 	:= 'Transport';

//Parameter setzen

ExecuteSkill.Parameter[3].ID := 3;
ExecuteSkill.Parameter[3].Name := 'Velocity';
ExecuteSkill.Parameter[3].Value := 300;



ExecuteSkill.Parameter[1].ID :=  1;
ExecuteSkill.Parameter[1].Name := 'TargetPosition X';
ExecuteSkill.Parameter[1].Value := 30 ;
ExecuteSkill.Parameter[1].StringValue := '#DP#2#XPosition';



ExecuteSkill.Parameter[2].ID := 2;
ExecuteSkill.Parameter[2].Name := 'TargetPosition Z';
ExecuteSkill.Parameter[2].Value := ZInputOutput;// ZCookieModule - ZCookieModuleCalibration - 2* Cookiethickness + toppingthickness+ Preasureheight  ;



(* ExecuteSkill.Parameter[4].ID := 4;
ExecuteSkill.Parameter[4].Name := 'Acceleration';
ExecuteSkill.Parameter[4].Value :=0 ;

*)
(*
ExecuteSkill.Parameter[5].ID := ;
ExecuteSkill.Parameter[5].Name := '';
ExecuteSkill.Parameter[5].Value := ;
*)



ExecuteSkill();

StepDone := ExecuteSkill.Done;
END_ACTION

ACTION Init_active:
//RT: 2014.11.23: Vorbereiten der daten und der HMI
RecipeDone := FALSE;

// Initialisation of Recipe Parameters an name etc
RecipeInfo.Name := 'Green Five';
RecipeInfo.Description := 'Remember spring feelings in autumn';
RecipeInfo.Dummy := FALSE;
RecipeInfo.RecipeID := 10057; 	// 
Initdone := TRUE;

//RT: 2014.11.23: wenn weniger als 5 alle lehren skills SkillID := 0
Command[1].SkillID := 1117;
Command[1].SkillName := 'Orange Juice';
Command[1].Quantity := 20;

Command[2].SkillID := 1112;
Command[2].SkillName := 'Lemon Juice';
Command[2].Quantity := 10;

Command[3].SkillID := 1114;
Command[3].SkillName := 'Pineapple Juice';
Command[3].Quantity := 30;

Command[4].SkillID := 1113;
Command[4].SkillName := 'Maracuja Juice';
Command[4].Quantity := 30;

Command[5].SkillID := 1119;
Command[5].SkillName := 'Blue Curacao';
Command[5].Quantity := 10;








//Parameter 0:

	RecipeInfo.UserParameter[0].Dummy 		:= FALSE;
	RecipeInfo.UserParameter[0].Default		:= 200;
	RecipeInfo.UserParameter[0].Description	:= 'Gives the total fluid amount in the glass';
	RecipeInfo.UserParameter[0].MaxValue	:= 200;
	RecipeInfo.UserParameter[0].MinValue	:= 10;
	RecipeInfo.UserParameter[0].Name		:= 'Total Liquid Amount';
	RecipeInfo.UserParameter[0].Unit		:= 'ml';
	
//Parameter 1-5:
FOR i := 1 TO 5 DO
	IF Command[i].SkillID = 0 THEN
		RecipeInfo.UserParameter[i].Dummy 		:= TRUE;
	ELSE
		RecipeInfo.UserParameter[i].Dummy 		:= FALSE;
		RecipeInfo.UserParameter[i].Default		:= Command[i].Quantity;
		RecipeInfo.UserParameter[i].Description	:= Command[i].SkillName;
		RecipeInfo.UserParameter[i].MaxValue	:= 100;
		RecipeInfo.UserParameter[i].MinValue	:= 1;
		RecipeInfo.UserParameter[i].Name		:= Command[i].SkillName;
		RecipeInfo.UserParameter[i].Unit		:= 'ml';	
	END_IF
END_FOR
END_ACTION

ACTION ST1_Input_active:
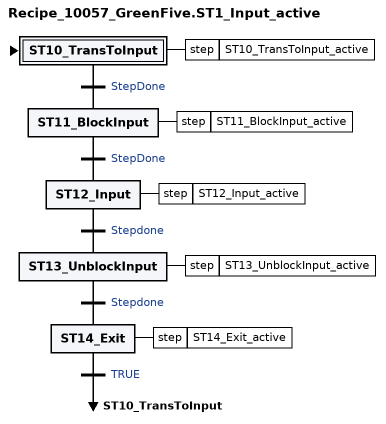
INITIAL_STEP ST10_TransToInput:
    ST10_TransToInput_active(N);  // step action
END_STEP
TRANSITION FROM ST10_TransToInput TO ST11_BlockInput
    := StepDone;
END_TRANSITION
STEP ST11_BlockInput:
    ST11_BlockInput_active(N);  // step action
END_STEP
TRANSITION FROM ST11_BlockInput TO ST12_Input
    := StepDone;
END_TRANSITION
STEP ST12_Input:
    ST12_Input_active(N);  // step action
END_STEP
TRANSITION FROM ST12_Input TO ST13_UnblockInput
    := Stepdone;
END_TRANSITION
STEP ST13_UnblockInput:
    ST13_UnblockInput_active(N);  // step action
END_STEP
TRANSITION FROM ST13_UnblockInput TO ST14_Exit
    := Stepdone;
END_TRANSITION
STEP ST14_Exit:
    ST14_Exit_active(N);  // step action
END_STEP
TRANSITION FROM ST14_Exit TO ST10_TransToInput
    := TRUE;
END_TRANSITION
END_ACTION

ACTION ST31_BlockPump_active:
//RT: 2014.11.23: Blockirt den Mover an Position
StepDone := FALSE;

//Skill auswählen
ExecuteSkill.SkillID 		:= 1315;
ExecuteSkill.SkillName	 	:= 'Block';

//Parameter setzen

ExecuteSkill.Parameter[1].ID := 1;
ExecuteSkill.Parameter[1].Name := 'TaskID';
ExecuteSkill.Parameter[1].Value := Order.TaskID;


(*
ExecuteSkill.Parameter[2].ID := ;
ExecuteSkill.Parameter[2].Name := '';
ExecuteSkill.Parameter[2].Value := ;
*)

(*
ExecuteSkill.Parameter[3].ID := ;
ExecuteSkill.Parameter[3].Name := '';
ExecuteSkill.Parameter[3].Value := ;
*)

(*
ExecuteSkill.Parameter[4].ID := ;
ExecuteSkill.Parameter[4].Name := '';
ExecuteSkill.Parameter[4].Value := ;
*)

(*
ExecuteSkill.Parameter[5].ID := ;
ExecuteSkill.Parameter[5].Name := '';
ExecuteSkill.Parameter[5].Value := ;
*)



ExecuteSkill();

StepDone := ExecuteSkill.Done;
END_ACTION

END_FUNCTION_BLOCK

// ---- POUs/FB_INIT_RECIPE.TcPOU
FUNCTION_BLOCK FB_INIT_RECIPE
VAR_INPUT
	Execute	: 	BOOL;
END_VAR
VAR_OUTPUT
	Done	: BOOL;
	Busy	: BOOL;
	Error	: BOOL;
END_VAR
VAR
	i	: INT := 10000;
	OfferCounter	: INT;
	InitOrder		: DUT_RECIPEORDER;
	fbExecuteRecipe	: FB_ExecuteRecipe;
	state: INT;
END_VAR

IF Execute THEN
	Done := FALSE;
	CASE state OF
		

		0: 
			fbExecuteRecipe.Execute := TRUE;
			InitOrder.RecipeID := i;
			state := 1;
			
		1:	
			fbExecuteRecipe(Order:= InitOrder);
			IF fbExecuteRecipe.Done THEN
				IF fbExecuteRecipe.NotAvailable THEN
				state := 50;
				ELSE
				Offer[OfferCounter]:=fbExecuteRecipe.RecipeInfo;
				OfferCounter := OfferCounter +1;
				state := 50;
				END_IF
			END_IF	
			
			
			
			
		50: IF i< 10100 THEN
				i := i+1;
				state :=0;
			ELSE
				busy 	:= FALSE;
				done 	:= TRUE;
				Execute := FALSE;
				state := 0;
			END_IF
		
		
		
		
		
		

	END_CASE
END_IF

END_FUNCTION_BLOCK

// ---- POUs/OPC/FB_ReadReset.TcPOU
FUNCTION_BLOCK FB_ReadReset
VAR_INPUT
	ReadIdentifier: STRING[80];
	NamespaceIndex: UINT;
	ConnectionHdl: DWORD;
	execute: BOOL;
END_VAR
VAR_OUTPUT
	ReadData		: BOOL;
	done: BOOL;
	busy: BOOL;
	error: BOOL;
END_VAR
VAR
		/// FBs
	fbNodeGetHandle: UA_NodeGetHandle;
	fbReadVariable: UA_Read;
	///Variables
	pReadData		: POINTER TO BOOL;
	
	VariableSize: UDINT;
	NodeHdl: DWORD;
	cbDataR: UDINT;
	state: INT := -1;
	SessionNodeID: ST_UANodeID;
	Timeout: TIME := DEFAULT_ADS_TIMEOUT;
END_VAR

IF execute THEN 
	DONE := FALSE;
	CASE state OF
		
		-1:	SessionNodeID.nNamespaceIndex    			:= Namespaceindex;
			SessionNodeID.eIdentifierType				:= 1;
			SessionNodeID.sIdentifier					:= ReadIdentifier;
			VariableSize 								:= SIZEOF (ReadData);
			pReadData									:= ADR(ReadData);
			
			
			

			busy := TRUE;
			done := FALSE;
			state:=0;

		0: fbNodeGetHandle(
			Execute:=FALSE,
			ConnectionHdl:=ConnectionHdl,
			NodeID:=SessionNodeID,
			Timeout:=Timeout,
			NodeHdl=>NodeHdl,
			Done=>,
			Busy=>busy,
			Error=>,
			ErrorID=>,);
			state:=1;
			
			
		1:fbNodeGetHandle(
			Execute:=TRUE,
			ConnectionHdl:=ConnectionHdl,
			NodeID:=SessionNodeID,
			Timeout:=Timeout,
			NodeHdl=>NodeHdl,
			Done=>,
			Busy=>busy,
			Error=>,
			ErrorID=>,);
			IF fbNodeGetHandle.Done THEN
			state := 2;
			END_IF
			IF fbNodeGetHandle.Error THEN
				state := -1;
			END_IF
		2:
			fbReadVariable(
				Execute:= FALSE, 
				ConnectionHdl:= ConnectionHdl, 
				NodeHdl:= NodeHdl, 
				stNodeAddInfo:= , 
				pVariable:= pReadData, 
				cbData:= VariableSize, 
				Timeout:= DEFAULT_ADS_TIMEOUT, 
				Done=> , 
				Busy=> , 
				Error=> , 
				ErrorID=> , 
				cbData_R=>cbDataR );
				state := 3;
				error :=FALSE;
				
		3:		fbReadVariable(
				Execute:= TRUE, 
				ConnectionHdl:= ConnectionHdl, 
				NodeHdl:= NodeHdl, 
				stNodeAddInfo:=, 
				pVariable:= pReadData, 
				cbData:= VariableSize, 
				Timeout:= DEFAULT_ADS_TIMEOUT, 
				Done=>, 
				Busy=>, 
				Error=>error, 
				ErrorID=>, 
				cbData_R=>cbDataR );
				IF fbReadVariable.Done THEN
					state		:= 2;
					execute		:= FALSE;
					done		:= TRUE;
					busy		:= FALSE;
				END_IF	
				IF fbReadVariable.Error THEN
				state := -1;
				END_IF	
		
	END_CASE
ELSE
	state := -1;
END_IF

END_FUNCTION_BLOCK

// ---- POUs/OPC/FB_WriteReset.TcPOU
FUNCTION_BLOCK FB_WriteReset
VAR_INPUT
	WriteIdentifier: STRING[80];
	NamespaceIndex: UINT;
	ConnectionHdl: DWORD;
	execute: BOOL;
	WriteData:  BOOL;
END_VAR
VAR_OUTPUT
	done: BOOL;
	busy: BOOL;
	error: BOOL;
END_VAR
VAR
	/// FBs
	fbWriteVariable: UA_Write;
	fbNodeGetHandle: UA_NodeGetHandle;
	fbNodeReleaseHandle	: UA_NodeReleaseHandle;
	/// Variables
	state: INT := -1;
	pWriteData: POINTER TO BOOL;
	VariableSize: UDINT;
	NodeHdl: DWORD;
	Timeout: TIME := DEFAULT_ADS_TIMEOUT;
	SessionNodeID: ST_UANodeID;
	Timer	: TON;
END_VAR

IF execute THEN
	Done := FALSE;
	CASE state OF
		
		-1:	SessionNodeID.nNamespaceIndex    			:= Namespaceindex;
			SessionNodeID.eIdentifierType				:= 1;
			SessionNodeID.sIdentifier					:= WriteIdentifier;
			VariableSize 								:= SIZEOF (WriteData);
			pWriteData									:= ADR(WriteData);
			
			
			done := FALSE;
			state:=0;
		
	    0: fbNodeGetHandle(
			Execute:=FALSE,
			ConnectionHdl:=ConnectionHdl,
			NodeID:=SessionNodeID,
			Timeout:=Timeout,
			NodeHdl=>NodeHdl,
			Done=>,
			Busy=>,
			Error=>,
			ErrorID=>,);
			state:=1;
			
		1:fbNodeGetHandle(
			Execute:=TRUE,
			ConnectionHdl:=ConnectionHdl,
			NodeID:=SessionNodeID,
			Timeout:=Timeout,
			NodeHdl=>NodeHdl,
			Done=>,
			Busy=>,
			Error=>,
			ErrorID=>,);
			IF fbNodeGetHandle.Done THEN
			state := 2;
			END_IF
			
		
				
		2: fbWriteVariable(
				Execute:=FALSE , 
				ConnectionHdl:=ConnectionHdl , 
				NodeHdl:=NodeHdl , 
				stNodeAddInfo:= , 
				pVariable:= pWriteData, 
				cbData:= VariableSize, 
				Timeout:=Timeout , 
				Done=> , 
				Busy=> , 
				Error=> , 
				ErrorID=> );
				
				state:=3;
				
		3: fbWriteVariable(
				Execute:=TRUE , 
				ConnectionHdl:=ConnectionHdl , 
				NodeHdl:=NodeHdl , 
				stNodeAddInfo:= , 
				pVariable:= pWriteData, 
				cbData:= VariableSize, 
				Timeout:=Timeout , 
				Done=> , 
				Busy=> , 
				Error=> , 
				ErrorID=> );
				IF fbWriteVariable.Done THEN
					state := 4;
				END_IF
				
		4: fbNodeReleaseHandle(ConnectionHdl := ConnectionHdl, Execute := FALSE, NodeHdl := NodeHdl, Timeout := Timeout);
			state := 5;
			Timer(IN := FALSE, PT := T#10S);
		5: 
			fbNodeReleaseHandle(ConnectionHdl := ConnectionHdl, Execute := TRUE, NodeHdl := NodeHdl, Timeout := Timeout);
				IF fbNodeReleaseHandle.Done OR Timer.Q THEN
					state		:= -1;
					execute		:= FALSE;
					done		:= TRUE;
					busy		:= FALSE;
				END_IF
			Timer(IN := TRUE);
			
				
	END_CASE
ELSE
	state := -1;
END_IF

END_FUNCTION_BLOCK

// ---- POUs/OPC/FB_OPCServerConnect.TcPOU
FUNCTION_BLOCK FB_OPCServerConnect
VAR_INPUT
	ServerUrl: STRING[80];
	NamespaceUri: STRING[80];
	ClientName: STRING[80];
	execute: BOOL;
END_VAR
VAR_OUTPUT
	ConnectHdl: DWORD;
	Namespaceindex: UINT;
	busy: BOOL;
	done: BOOL;
	error: BOOL;
END_VAR
VAR
	fbGetNameSpace: UA_GetNameSpaceIndex;
	SessionconnectInfo: ST_UASessionConnectInfo;
	Timeout: TIME := DEFAULT_ADS_TIMEOUT;
	state: INT := -1;
	fbConnect: UA_Connect;
END_VAR

IF execute THEN
	CASE state OF
	-1: 	SessionconnectInfo.sApplicationName			:=ClientName;
			SessionconnectInfo.eSecurityMode				:=1; 
			SessionconnectInfo.eSecurityPolicyUri		:=1;
			SessionconnectInfo.eTransportProfileUri		:=1;
			SessionconnectInfo.tConnectTimeout			:=T#4S;
			SessionconnectInfo.tSessionTimeout			:=T#3S;
			
			
			busy 	:= TRUE;
			done	:= FALSE;							
			state 	:= 0;

	0:
         fbConnect(
			Execute:= FALSE, 
			ServerUrl:=ServerUrl , 
			SessionConnectInfo:= SessionconnectInfo, 
			Timeout:= Timeout, 
			ConnectionHdl=> ConnectHdl, 
			Done=>, 
			Busy=>busy, 
			Error=>error, 
			ErrorID=>);
			
	 		state := 1;
			
	1:
         fbConnect(
			Execute:= TRUE, 
			ServerUrl:=ServerUrl , 
			SessionConnectInfo:= SessionconnectInfo, 
			Timeout:= Timeout, 
			ConnectionHdl=> ConnectHdl,  
			Done=>, 
			Busy=>busy, 
			Error=>error, 
			ErrorID=> );
			
			IF fbConnect.done THEN
			
			state := 2;
			END_IF
			
			IF fbConnect.Error THEN
				error := TRUE;
			state := 0;
			END_IF
		

			
 		
		
	2:	
		fbGetNameSpace(
			Execute:= FALSE,
			ConnectionHdl:=ConnectHdl,
			NamespaceUri:=NamespaceUri,
			Timeout:=Timeout,
			NamespaceIndex=>Namespaceindex,
			Done=>,
			Busy=>busy,
			Error=>error,
			ErrorID=>,);	
			
			state := 3;	
	3:
		fbGetNameSpace(
			Execute:= TRUE,
			ConnectionHdl:=ConnectHdl,
			NamespaceUri:=NamespaceUri,
			Timeout:=Timeout,
			NamespaceIndex=>Namespaceindex,
			Done=>,
			Busy=>busy,
			Error=>error,
			ErrorID=>,);
			IF fbGetNameSpace.done THEN
			Execute := FALSE;
			busy	:= FALSE;
			done	:= TRUE;
			state 	:= 0;
			END_IF
		END_CASE
ELSE
	done	:= FALSE;
	busy := FALSE;
	error := FALSE;
	state := -1;
END_IF

END_FUNCTION_BLOCK

// ---- POUs/OPC/FB_WriteOfferlist.TcPOU
FUNCTION_BLOCK FB_WriteOfferlist
VAR_INPUT
	WriteIdentifier: STRING[80];
	NamespaceIndex: UINT;
	ConnectionHdl: DWORD;
	execute: BOOL;
	WriteData:  ARRAY [0..OfferCnt] OF DUT_RECIPEOFFER;
END_VAR
VAR_OUTPUT
	done: BOOL;
	busy: BOOL;
	error: BOOL;
END_VAR
VAR
	/// FBs
	fbWriteVariable: UA_Write;
	fbNodeGetHandle: UA_NodeGetHandle;
	/// Variables
	state: INT := -1;
	pWriteData: POINTER TO DUT_RECIPEOFFER;
	VariableSize: UDINT;
	NodeHdl: DWORD;
	Timeout: TIME := DEFAULT_ADS_TIMEOUT;
	SessionNodeID: ST_UANodeID;
END_VAR

IF execute THEN
	CASE state OF
		
		-1:	SessionNodeID.nNamespaceIndex    			:= Namespaceindex;
			SessionNodeID.eIdentifierType				:= 1;
			SessionNodeID.sIdentifier					:= WriteIdentifier;
			VariableSize 								:= SIZEOF (WriteData);
			pWriteData								:= ADR(WriteData);
			
			
			done := FALSE;
			state:=0;
		
	    0: fbNodeGetHandle(
			Execute:=FALSE,
			ConnectionHdl:=ConnectionHdl,
			NodeID:=SessionNodeID,
			Timeout:=Timeout,
			NodeHdl=>NodeHdl,
			Done=>,
			Busy=>,
			Error=>,
			ErrorID=>,);
			state:=1;
			
		1:fbNodeGetHandle(
			Execute:=TRUE,
			ConnectionHdl:=ConnectionHdl,
			NodeID:=SessionNodeID,
			Timeout:=Timeout,
			NodeHdl=>NodeHdl,
			Done=>,
			Busy=>,
			Error=>,
			ErrorID=>,);
			IF fbNodeGetHandle.Done THEN
			state := 2;
			END_IF
			
		
				
		2: fbWriteVariable(
				Execute:=FALSE , 
				ConnectionHdl:=ConnectionHdl , 
				NodeHdl:=NodeHdl , 
				stNodeAddInfo:= , 
				pVariable:= pWriteData, 
				cbData:= VariableSize, 
				Timeout:=Timeout , 
				Done=> , 
				Busy=> , 
				Error=> , 
				ErrorID=> );
				
				state:=3;
				
		3: fbWriteVariable(
				Execute:=TRUE , 
				ConnectionHdl:=ConnectionHdl , 
				NodeHdl:=NodeHdl , 
				stNodeAddInfo:= , 
				pVariable:= pWriteData, 
				cbData:= VariableSize, 
				Timeout:=Timeout , 
				Done=> , 
				Busy=> , 
				Error=> , 
				ErrorID=> );
				IF fbWriteVariable.Done THEN
					state		:= 2;
					execute		:= FALSE;
					done		:= TRUE;
					busy		:= FALSE;
				END_IF		
	END_CASE
ELSE
	state := -1;
END_IF

END_FUNCTION_BLOCK

// ---- POUs/OPC/FB_ReadQueue.TcPOU
FUNCTION_BLOCK FB_ReadQueue
VAR_INPUT
	ReadIdentifier: STRING[80];
	NamespaceIndex: UINT;
	ConnectionHdl: DWORD;
	execute: BOOL;
END_VAR
VAR_OUTPUT
	ReadData		: DUT_RECIPEORDER;
	done: BOOL;
	busy: BOOL;
	error: BOOL;
END_VAR
VAR
		/// FBs
	fbNodeGetHandle: UA_NodeGetHandle;
	fbReadVariable: UA_Read;
	///Variables
	pReadData		: POINTER TO DUT_RECIPEORDER;
	
	VariableSize: UDINT;
	NodeHdl: DWORD;
	cbDataR: UDINT;
	state: INT := -1;
	SessionNodeID: ST_UANodeID;
	Timeout: TIME := DEFAULT_ADS_TIMEOUT;
END_VAR

IF execute THEN 
	DONE := FALSE;
	CASE state OF
		
		-1:	SessionNodeID.nNamespaceIndex    			:= Namespaceindex;
			SessionNodeID.eIdentifierType				:= 1;
			SessionNodeID.sIdentifier					:= ReadIdentifier;
			VariableSize 								:= SIZEOF (ReadData);
			pReadData									:= ADR(ReadData);
			
			
			

			busy := TRUE;
			done := FALSE;
			state:=0;

		0: fbNodeGetHandle(
			Execute:=FALSE,
			ConnectionHdl:=ConnectionHdl,
			NodeID:=SessionNodeID,
			Timeout:=Timeout,
			NodeHdl=>NodeHdl,
			Done=>,
			Busy=>busy,
			Error=>,
			ErrorID=>,);
			state:=1;
			
		1:fbNodeGetHandle(
			Execute:=TRUE,
			ConnectionHdl:=ConnectionHdl,
			NodeID:=SessionNodeID,
			Timeout:=Timeout,
			NodeHdl=>NodeHdl,
			Done=>,
			Busy=>busy,
			Error=>,
			ErrorID=>,);
			IF fbNodeGetHandle.Done THEN
			state := 2;
			END_IF
			
		2:
			fbReadVariable(
				Execute:= FALSE, 
				ConnectionHdl:= ConnectionHdl, 
				NodeHdl:= NodeHdl, 
				stNodeAddInfo:= , 
				pVariable:= pReadData, 
				cbData:= VariableSize, 
				Timeout:= DEFAULT_ADS_TIMEOUT, 
				Done=> , 
				Busy=> , 
				Error=> , 
				ErrorID=> , 
				cbData_R=>cbDataR );
				state := 3;
				error :=FALSE;
				
		3:		fbReadVariable(
				Execute:= TRUE, 
				ConnectionHdl:= ConnectionHdl, 
				NodeHdl:= NodeHdl, 
				stNodeAddInfo:=, 
				pVariable:= pReadData, 
				cbData:= VariableSize, 
				Timeout:= DEFAULT_ADS_TIMEOUT, 
				Done=>, 
				Busy=>, 
				Error=>error, 
				ErrorID=>, 
				cbData_R=>cbDataR );
				IF fbReadVariable.Done THEN
					state		:= 2;
					execute		:= FALSE;
					done		:= TRUE;
					busy		:= FALSE;
				END_IF		
		
	END_CASE
ELSE
	state := -1;
END_IF

END_FUNCTION_BLOCK

// ---- POUs/OPC/FB_WriteTask.TcPOU
FUNCTION_BLOCK FB_WriteTask
VAR_INPUT
	WriteIdentifier: STRING[80];
	NamespaceIndex: UINT;
	ConnectionHdl: DWORD;
	execute: BOOL;
	WriteData:  DUT_TASK;
END_VAR
VAR_OUTPUT
	done: BOOL;
	busy: BOOL;
	error: BOOL;
END_VAR
VAR
	/// FBs
	fbWriteVariable: UA_Write;
	fbNodeGetHandle: UA_NodeGetHandle;
	/// Variables
	state: INT := -1;
	pWriteData: POINTER TO DUT_TASK;
	VariableSize: UDINT;
	NodeHdl: DWORD;
	Timeout: TIME := DEFAULT_ADS_TIMEOUT;
	SessionNodeID: ST_UANodeID;
END_VAR

IF execute THEN
	DONE := FALSE;
	CASE state OF
		
		-1:	SessionNodeID.nNamespaceIndex    			:= Namespaceindex;
			SessionNodeID.eIdentifierType				:= 1;
			SessionNodeID.sIdentifier					:= WriteIdentifier;
			VariableSize 								:= SIZEOF (WriteData);
			pWriteData								:= ADR(WriteData);
			
			
			done := FALSE;
			state:=0;
		
	    0: fbNodeGetHandle(
			Execute:=FALSE,
			ConnectionHdl:=ConnectionHdl,
			NodeID:=SessionNodeID,
			Timeout:=Timeout,
			NodeHdl=>NodeHdl,
			Done=>,
			Busy=>,
			Error=>,
			ErrorID=>,);
			state:=1;
			
		1:fbNodeGetHandle(
			Execute:=TRUE,
			ConnectionHdl:=ConnectionHdl,
			NodeID:=SessionNodeID,
			Timeout:=Timeout,
			NodeHdl=>NodeHdl,
			Done=>,
			Busy=>,
			Error=>,
			ErrorID=>,);
			IF fbNodeGetHandle.Done THEN
			state := 2;
			END_IF
			
		
				
		2: fbWriteVariable(
				Execute:=FALSE , 
				ConnectionHdl:=ConnectionHdl , 
				NodeHdl:=NodeHdl , 
				stNodeAddInfo:= , 
				pVariable:= pWriteData, 
				cbData:= VariableSize, 
				Timeout:=Timeout , 
				Done=> , 
				Busy=> , 
				Error=> , 
				ErrorID=> );
				
				state:=3;
				
		3: fbWriteVariable(
				Execute:=TRUE , 
				ConnectionHdl:=ConnectionHdl , 
				NodeHdl:=NodeHdl , 
				stNodeAddInfo:= , 
				pVariable:= pWriteData, 
				cbData:= VariableSize, 
				Timeout:=Timeout , 
				Done=> , 
				Busy=> , 
				Error=> , 
				ErrorID=> );
				IF fbWriteVariable.Done THEN
					state		:= -1;
					execute		:= FALSE;
					done		:= TRUE;
					busy		:= FALSE;
				END_IF		
	END_CASE
ELSE
	state := -1;
END_IF

END_FUNCTION_BLOCK

// ---- POUs/OPC/FB_WriteQueue.TcPOU
FUNCTION_BLOCK FB_WriteQueue
VAR_INPUT
	WriteIdentifier: STRING[80];
	NamespaceIndex: UINT;
	ConnectionHdl: DWORD;
	execute: BOOL;
	WriteData:  DUT_RECIPEORDER;
END_VAR
VAR_OUTPUT
	done: BOOL;
	busy: BOOL;
	error: BOOL;
END_VAR
VAR
	/// FBs
	fbWriteVariable: UA_Write;
	fbNodeGetHandle: UA_NodeGetHandle;
	fbNodeReleaseHandle	: UA_NodeReleaseHandle;
	/// Variables
	state: INT := -1;
	pWriteData: POINTER TO DUT_RECIPEORDER;
	VariableSize: UDINT;
	NodeHdl: DWORD;
	Timeout: TIME := DEFAULT_ADS_TIMEOUT;
	SessionNodeID: ST_UANodeID;
END_VAR

IF execute THEN
	Done := FALSE;
	CASE state OF
		
		-1:	SessionNodeID.nNamespaceIndex    			:= Namespaceindex;
			SessionNodeID.eIdentifierType				:= 1;
			SessionNodeID.sIdentifier					:= WriteIdentifier;
			VariableSize 								:= SIZEOF (WriteData);
			pWriteData								:= ADR(WriteData);
			
			
			done := FALSE;
			state:=0;
		
	    0: fbNodeGetHandle(
			Execute:=FALSE,
			ConnectionHdl:=ConnectionHdl,
			NodeID:=SessionNodeID,
			Timeout:=Timeout,
			NodeHdl=>NodeHdl,
			Done=>,
			Busy=>,
			Error=>,
			ErrorID=>,);
			state:=1;
			
		1:fbNodeGetHandle(
			Execute:=TRUE,
			ConnectionHdl:=ConnectionHdl,
			NodeID:=SessionNodeID,
			Timeout:=Timeout,
			NodeHdl=>NodeHdl,
			Done=>,
			Busy=>,
			Error=>,
			ErrorID=>,);
			IF fbNodeGetHandle.Done THEN
			state := 2;
			END_IF
			
		
				
		2: fbWriteVariable(
				Execute:=FALSE , 
				ConnectionHdl:=ConnectionHdl , 
				NodeHdl:=NodeHdl , 
				stNodeAddInfo:= , 
				pVariable:= pWriteData, 
				cbData:= VariableSize, 
				Timeout:=Timeout , 
				Done=> , 
				Busy=> , 
				Error=> , 
				ErrorID=> );
				
				state:=3;
				
		3: fbWriteVariable(
				Execute:=TRUE , 
				ConnectionHdl:=ConnectionHdl , 
				NodeHdl:=NodeHdl , 
				stNodeAddInfo:= , 
				pVariable:= pWriteData, 
				cbData:= VariableSize, 
				Timeout:=Timeout , 
				Done=> , 
				Busy=> , 
				Error=> , 
				ErrorID=> );
				IF fbWriteVariable.Done THEN
					state := 4;
				END_IF
				
		4: fbNodeReleaseHandle(ConnectionHdl := ConnectionHdl, Execute := FALSE, NodeHdl := NodeHdl, Timeout := Timeout);
			state := 5;
		5: fbNodeReleaseHandle(ConnectionHdl := ConnectionHdl, Execute := TRUE, NodeHdl := NodeHdl, Timeout := Timeout);
				IF fbNodeReleaseHandle.Done THEN
					state		:= -1;
					execute		:= FALSE;
					done		:= TRUE;
					busy		:= FALSE;
				END_IF		
	END_CASE
ELSE
	state := -1;
END_IF

END_FUNCTION_BLOCK

// ---- POUs/FB_AddSkill.TcPOU
FUNCTION_BLOCK FB_AddSkill
VAR_INPUT
	SkillID 		: UINT;
	SkillName		: STRING[80];
    Parameter 		: ARRAY [0..ParameterCnt] OF DUT_PARAMETER;
	EmptyParameter	: ARRAY [0..ParameterCnt] OF DUT_PARAMETER;
	TargetSkillNo	: INT := 0;
	
END_VAR
VAR_OUTPUT
	Done			: BOOL;
END_VAR
VAR
	
	
	i: INT;
END_VAR

DONE := FALSE;

	
	
	
	TempTask.Skill[TargetSkillNo].Dummy 	:= FALSE;
	TempTask.Skill[TargetSkillNo].ID 		:= SkillID;
	TempTask.Skill[TargetSkillNo].Name	:= SkillName;
	
	FOR i := 0 TO ParameterCnt DO
		IF NOT (Parameter[i].ID = 0) THEN
			TempTask.Skill[TargetSkillNo].Parameter[i].Dummy 	:= FALSE;
			TempTask.Skill[TargetSkillNo].Parameter[i].Value	:= Parameter[i].Value;
			TempTask.Skill[TargetSkillNo].Parameter[i].StringValue	:= Parameter[i].StringValue;
			TempTask.Skill[TargetSkillNo].Parameter[i].ID 	:= Parameter[i].ID;
			TempTask.Skill[TargetSkillNo].Parameter[i].Name	:= Parameter[i].Name;
			
		END_IF
	END_FOR
	
	//Mitzählen, welche stelle der Taskskillliste gerade befüllt wird
	TargetSkillNo := TargetSkillNo +1;
	Parameter := EmptyParameter;
Done := TRUE;

END_FUNCTION_BLOCK

// ---- POUs/OPC/FB_ReadRecipeTool.TcPOU
FUNCTION_BLOCK FB_ReadRecipeTool
VAR_INPUT
	ReadIdentifier: STRING[80];
	NamespaceIndex: UINT;
	ConnectionHdl: DWORD;
	execute: BOOL;
END_VAR
VAR_OUTPUT
	OrderRead		: ARRAY [1..OrderCnt] OF DUT_RECIPEORDER;
	done: BOOL;
	busy: BOOL;
	error: BOOL;
END_VAR
VAR
		/// FBs
	fbNodeGetHandle: UA_NodeGetHandle;
	fbReadVariable: UA_Read;
	///Variables
	pOrderInput		: POINTER TO ARRAY [1..OrderCnt] OF DUT_RECIPEORDER;
	
	VariableSize: UDINT;
	NodeHdl: DWORD;
	cbDataR: UDINT;
	state: INT := -1;
	SessionNodeID: ST_UANodeID;
	Timeout: TIME := DEFAULT_ADS_TIMEOUT;
END_VAR

IF execute THEN 
	CASE state OF
		
		-1:	SessionNodeID.nNamespaceIndex    			:= Namespaceindex;
			SessionNodeID.eIdentifierType				:= 1;
			SessionNodeID.sIdentifier					:= ReadIdentifier;
			VariableSize 								:= SIZEOF (OrderInput);
			pOrderInput								:= ADR(OrderInput);
			
			
			

			busy := TRUE;
			done := FALSE;
			state:=0;

		0: fbNodeGetHandle(
			Execute:=FALSE,
			ConnectionHdl:=ConnectionHdl,
			NodeID:=SessionNodeID,
			Timeout:=Timeout,
			NodeHdl=>NodeHdl,
			Done=>,
			Busy=>busy,
			Error=>,
			ErrorID=>,);
			state:=1;
			
		1:fbNodeGetHandle(
			Execute:=TRUE,
			ConnectionHdl:=ConnectionHdl,
			NodeID:=SessionNodeID,
			Timeout:=Timeout,
			NodeHdl=>NodeHdl,
			Done=>,
			Busy=>busy,
			Error=>,
			ErrorID=>,);
			IF fbNodeGetHandle.Done THEN
			state := 2;
			END_IF
			
		2:
			fbReadVariable(
				Execute:= FALSE, 
				ConnectionHdl:= ConnectionHdl, 
				NodeHdl:= NodeHdl, 
				stNodeAddInfo:= , 
				pVariable:= pOrderInput, 
				cbData:= VariableSize, 
				Timeout:= DEFAULT_ADS_TIMEOUT, 
				Done=> , 
				Busy=> , 
				Error=> , 
				ErrorID=> , 
				cbData_R=>cbDataR );
				state := 3;
				error :=FALSE;
				
		3:		fbReadVariable(
				Execute:= TRUE, 
				ConnectionHdl:= ConnectionHdl, 
				NodeHdl:= NodeHdl, 
				stNodeAddInfo:=, 
				pVariable:= pOrderInput, 
				cbData:= VariableSize, 
				Timeout:= DEFAULT_ADS_TIMEOUT, 
				Done=>, 
				Busy=>, 
				Error=>error, 
				ErrorID=>, 
				cbData_R=>cbDataR );
				IF fbReadVariable.Done THEN
					state		:= 2;
					execute		:= FALSE;
					done		:= TRUE;
					busy		:= FALSE;
				END_IF		
		
	END_CASE
 
END_IF

END_FUNCTION_BLOCK

// ---- POUs/OPC/FB_UpdateRecipeTool.TcPOU
FUNCTION_BLOCK FB_UpdateRecipeTool
VAR_INPUT
	ServerUrl		: STRING[80];
	NamespaceUri	: STRING[80];
	ClientName		: STRING[80];
	IdentifierInput	: STRING[80];
	IdentifierOutput: STRING[80];
	Execute			: BOOL;
	
END_VAR
VAR_OUTPUT
	RecipeToolRead		: ARRAY [1..OrderCnt] OF DUT_RECIPEORDER;
	done				: BOOL := FALSE;
	connected			: BOOL := FALSE;
	readestablished		: BOOL := FALSE;
	writedone			: BOOL := FALSE;
END_VAR
VAR
	fbConnect		: FB_OPCServerConnect;
	fbRead			: FB_ReadRecipeTool;
	fbWrite			: FB_WriteRecipeTool;
	NamespaceIndex	: UINT;
	ConnectionHdl	: DWORD;
	state: INT;
END_VAR

IF Execute THEN	

CASE state OF
	
	0: state := 1;
	1: fbConnect(
			ServerUrl:= ServerUrl, 
			NamespaceUri:= NamespaceUri , 
			ClientName:= ClientName , 
			execute:= TRUE, 
			ConnectHdl=> ConnectionHdl , 
			Namespaceindex=> NamespaceIndex , 
			busy=> , 
			done=> , 
			error=> );
		IF fbConnect.done THEN
		state := 2;
		END_IF
		
		
		
	
	2: fbRead(
			IdentifierInput:= IdentifierInput, 
			NamespaceIndex:= NamespaceIndex, 
			ConnectionHdl:= ConnectionHdl, 
			execute:= TRUE, 
			OrderInput=> OrderInput, 
			done=> done, 
			busy=> , 
			error=> );
		IF fbRead.done THEN
			writedone := TRUE;
		END_IF
		//state := 3;

			
	(*3:fbWrite(
		IdentifierOutput:= IdentifierOutput, 
		NamespaceIndex:= NamespaceIndex, 
		ConnectionHdl:= ConnectionHdl, 
		execute:= TRUE, 
		ModuleOutput:= ModuleOutput, 
		done=> , 
		busy=> , 
		error=> );
		
		state := 2;*)
		
		
	
		
		
END_CASE

END_IF

END_FUNCTION_BLOCK

// ---- POUs/Recipes/Recipe_10018_TripleCookiemitTopping.TcPOU
FUNCTION_BLOCK Recipe_10018_TripleCookiemitTopping
VAR_INPUT
	execute	: BOOL;
	Order	: DUT_RECIPEORDER;
END_VAR
VAR_OUTPUT
	RecipeInfo	: DUT_RECIPEOFFER;
	RecipeDone	: BOOL;	
	InitDone	: BOOL;
END_VAR
VAR
	StepDone	: BOOL;
	Layercnt	: INT := 0;
	OrderLayers	: INT := 2;
	i : INT;
END_VAR

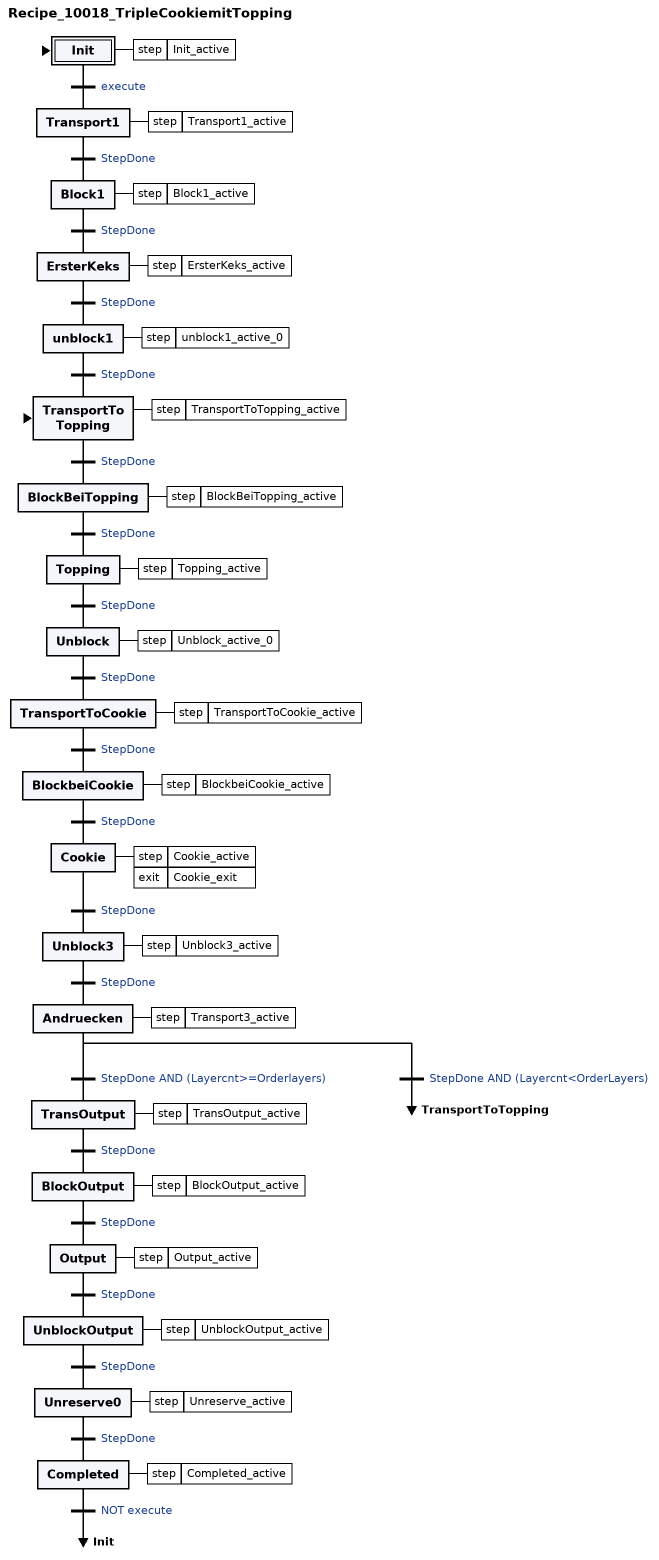
INITIAL_STEP Init:
    Init_active(N);  // step action
END_STEP
TRANSITION FROM Init TO Transport1
    := execute;
END_TRANSITION
STEP Transport1:
    Transport1_active(N);  // step action
END_STEP
TRANSITION FROM Transport1 TO Block1
    := StepDone;
END_TRANSITION
STEP Block1:
    Block1_active(N);  // step action
END_STEP
TRANSITION FROM Block1 TO ErsterKeks
    := StepDone;
END_TRANSITION
STEP ErsterKeks:
    ErsterKeks_active(N);  // step action
END_STEP
TRANSITION FROM ErsterKeks TO unblock1
    := StepDone;
END_TRANSITION
STEP unblock1:
    unblock1_active_0(N);  // step action
END_STEP
TRANSITION FROM unblock1 TO TransportToTopping
    := StepDone;
END_TRANSITION
STEP TransportToTopping:
    TransportToTopping_active(N);  // step action
END_STEP
TRANSITION FROM TransportToTopping TO BlockBeiTopping
    := StepDone;
END_TRANSITION
STEP BlockBeiTopping:
    BlockBeiTopping_active(N);  // step action
END_STEP
TRANSITION FROM BlockBeiTopping TO Topping
    := StepDone;
END_TRANSITION
STEP Topping:
    Topping_active(N);  // step action
END_STEP
TRANSITION FROM Topping TO Unblock
    := StepDone;
END_TRANSITION
STEP Unblock:
    Unblock_active_0(N);  // step action
END_STEP
TRANSITION FROM Unblock TO TransportToCookie
    := StepDone;
END_TRANSITION
STEP TransportToCookie:
    TransportToCookie_active(N);  // step action
END_STEP
TRANSITION FROM TransportToCookie TO BlockbeiCookie
    := StepDone;
END_TRANSITION
STEP BlockbeiCookie:
    BlockbeiCookie_active(N);  // step action
END_STEP
TRANSITION FROM BlockbeiCookie TO Cookie
    := StepDone;
END_TRANSITION
STEP Cookie:
    Cookie_active(N);  // step action
    Cookie_exit(P0);  // exit action
END_STEP
TRANSITION FROM Cookie TO Unblock3
    := StepDone;
END_TRANSITION
STEP Unblock3:
    Unblock3_active(N);  // step action
END_STEP
TRANSITION FROM Unblock3 TO Andruecken
    := StepDone;
END_TRANSITION
STEP Andruecken:
    Transport3_active(N);  // step action
END_STEP
TRANSITION FROM Andruecken TO TransOutput
    := StepDone AND (Layercnt>=Orderlayers);
END_TRANSITION
STEP TransOutput:
    TransOutput_active(N);  // step action
END_STEP
TRANSITION FROM TransOutput TO BlockOutput
    := StepDone;
END_TRANSITION
STEP BlockOutput:
    BlockOutput_active(N);  // step action
END_STEP
TRANSITION FROM BlockOutput TO Output
    := StepDone;
END_TRANSITION
STEP Output:
    Output_active(N);  // step action
END_STEP
TRANSITION FROM Output TO UnblockOutput
    := StepDone;
END_TRANSITION
STEP UnblockOutput:
    UnblockOutput_active(N);  // step action
END_STEP
TRANSITION FROM UnblockOutput TO Unreserve0
    := StepDone;
END_TRANSITION
TRANSITION FROM Andruecken TO TransportToTopping
    := StepDone AND (Layercnt<OrderLayers);
END_TRANSITION
STEP Unreserve0:
    Unreserve_active(N);  // step action
END_STEP
TRANSITION FROM Unreserve0 TO Completed
    := StepDone;
END_TRANSITION
STEP Completed:
    Completed_active(N);  // step action
END_STEP
TRANSITION FROM Completed TO Init
    := NOT execute;
END_TRANSITION

ACTION BlockOutput_active:
StepDone := FALSE;

//Skill auswählen



ExecuteSkill.SkillID 		:= 1315;
ExecuteSkill.SkillName	 	:= 'Block';

ExecuteSkill();

StepDone := ExecuteSkill.Done;
END_ACTION

ACTION Production2_active:
StepDone := FALSE;
RecipeDone := FALSE;
//Skill auswählen
ExecuteSkill.SkillID 		:= 1339;
ExecuteSkill.SkillName	 	:= 'ParameterTESTSKILL1339';


ExecuteSkill.Parameter[0].ID := 10;
ExecuteSkill.Parameter[0].Name := 'Blinkfrequenz';
ExecuteSkill.Parameter[0].Value := Order.UserParameter[0].Value*2;


ExecuteSkill();

StepDone := ExecuteSkill.Done;
END_ACTION

ACTION TransportToCookie_active:
StepDone := FALSE;

//Skill auswählen
ExecuteSkill.SkillID 		:= 1320;
ExecuteSkill.SkillName	 	:= 'Transport';

//Parameter setzen

ExecuteSkill.Parameter[3].ID := 3;
ExecuteSkill.Parameter[3].Name := 'Velocity';
ExecuteSkill.Parameter[3].Value := 400;



ExecuteSkill.Parameter[1].ID :=  1;
ExecuteSkill.Parameter[1].Name := 'TargetPosition X';
ExecuteSkill.Parameter[1].Value := 30 ;
ExecuteSkill.Parameter[1].StringValue := '#DP#2#XPosition';



ExecuteSkill.Parameter[2].ID := 2;
ExecuteSkill.Parameter[2].Name := 'TargetPosition Z';
ExecuteSkill.Parameter[2].Value := ZCookieModule + ZCookieModuleCalibration - ((Layercnt +1) * ( toppingthickness - cookiethickness)) ;

ExecuteSkill();

StepDone := ExecuteSkill.Done;
END_ACTION

ACTION Topping_active:
StepDone := FALSE;

//Skill auswählen
CASE REAL_TO_INT (order.UserParameter[2*LayerCnt].Value) OF
	1: 
		ExecuteSkill.SkillID 		:=  1230;
		ExecuteSkill.SkillName	 	:= 'Strawberry Topping';
	2: 
		ExecuteSkill.SkillID 		:=  1240;
		ExecuteSkill.SkillName	 	:= 'Apple Topping';
	ELSE
		ExecuteSkill.SkillID 		:=  1230;
		ExecuteSkill.SkillName	 	:= 'Strawberry Topping';
END_CASE


//Parameter setzen

ExecuteSkill.Parameter[0].ID := 1;
ExecuteSkill.Parameter[0].Name := 'Amount';
ExecuteSkill.Parameter[0].Value := order.UserParameter[2*LayerCnt + 1].Value ;


(*
ExecuteSkill.Parameter[1].ID := 1;
ExecuteSkill.Parameter[1].Name := 'TaskID';
ExecuteSkill.Parameter[1].Value := 130;
*)
(*
ExecuteSkill.Parameter[2].ID := ;
ExecuteSkill.Parameter[2].Name := '';
ExecuteSkill.Parameter[2].Value := ;
*)

(*
ExecuteSkill.Parameter[3].ID := ;
ExecuteSkill.Parameter[3].Name := '';
ExecuteSkill.Parameter[3].Value := ;
*)

(*
ExecuteSkill.Parameter[4].ID := ;
ExecuteSkill.Parameter[4].Name := '';
ExecuteSkill.Parameter[4].Value := ;
*)

(*
ExecuteSkill.Parameter[5].ID := ;
ExecuteSkill.Parameter[5].Name := '';
ExecuteSkill.Parameter[5].Value := ;
*)

ExecuteSkill();

StepDone := ExecuteSkill.Done;
END_ACTION

ACTION BlockbeiCookie_active:
StepDone := FALSE;

//Skill auswählen
ExecuteSkill.SkillID 		:= 1315;
ExecuteSkill.SkillName	 	:= 'Block';

//Parameter setzen

ExecuteSkill.Parameter[1].ID := 1;
ExecuteSkill.Parameter[1].Name := 'TaskID';
ExecuteSkill.Parameter[1].Value := 130;


(*
ExecuteSkill.Parameter[2].ID := ;
ExecuteSkill.Parameter[2].Name := '';
ExecuteSkill.Parameter[2].Value := ;
*)

(*
ExecuteSkill.Parameter[3].ID := ;
ExecuteSkill.Parameter[3].Name := '';
ExecuteSkill.Parameter[3].Value := ;
*)

(*
ExecuteSkill.Parameter[4].ID := ;
ExecuteSkill.Parameter[4].Name := '';
ExecuteSkill.Parameter[4].Value := ;
*)

(*
ExecuteSkill.Parameter[5].ID := ;
ExecuteSkill.Parameter[5].Name := '';
ExecuteSkill.Parameter[5].Value := ;
*)



ExecuteSkill();

StepDone := ExecuteSkill.Done;
END_ACTION

ACTION Unblock1_active:
StepDone := FALSE;

//Skill auswählen

CASE LREAL_TO_INT (order.UserParameter[2].Value) OF

1:
ExecuteSkill.SkillID 		:= 1316;
ExecuteSkill.SkillName	 	:= 'Unblock';

ExecuteSkill();

StepDone := ExecuteSkill.Done;
ELSE StepDone := TRUE;

END_CASE
END_ACTION

ACTION Transport_active:
StepDone := FALSE;

//Skill auswählen

CASE LREAL_TO_INT (order.UserParameter[2].Value) OF

1:
//Skill auswählen
ExecuteSkill.SkillID 		:= 1320;
ExecuteSkill.SkillName	 	:= 'Transport';

//Parameter setzen

ExecuteSkill.Parameter[3].ID :=3 ;
ExecuteSkill.Parameter[3].Name := 'Velocity';
ExecuteSkill.Parameter[3].Value := 1500;



ExecuteSkill.Parameter[1].ID :=1 ;
ExecuteSkill.Parameter[1].Name := 'TargetPosition X';
ExecuteSkill.Parameter[1].StringValue := '#DP#2#XPosition';
ExecuteSkill.Parameter[1].Value := 200 ;


ExecuteSkill.Parameter[2].ID := 2 ;
ExecuteSkill.Parameter[2].Name := 'TargetPosition Z';
ExecuteSkill.Parameter[2].Value := 90 ;



ExecuteSkill.Parameter[4].ID := 4 ;
ExecuteSkill.Parameter[4].Name := 'Acceleration';
ExecuteSkill.Parameter[4].Value := 4500;


(*
ExecuteSkill.Parameter[5].ID := ;
ExecuteSkill.Parameter[5].Name := '';
ExecuteSkill.Parameter[5].Value := ;
*)



ExecuteSkill();

StepDone := ExecuteSkill.Done;
ELSE StepDone := TRUE;

END_CASE
END_ACTION

ACTION Transport2_active:
StepDone := FALSE;

//Skill auswählen
ExecuteSkill.SkillID 		:= 1320;
ExecuteSkill.SkillName	 	:= 'Transport';

//Parameter setzen

ExecuteSkill.Parameter[3].ID := 3;
ExecuteSkill.Parameter[3].Name := 'Velocity';
ExecuteSkill.Parameter[3].Value := 2800;



ExecuteSkill.Parameter[1].ID :=  1;
ExecuteSkill.Parameter[1].Name := 'TargetPosition X';
ExecuteSkill.Parameter[1].Value := 30 ;
ExecuteSkill.Parameter[1].StringValue := '#DP#2#XPosition';



ExecuteSkill.Parameter[2].ID := 2;
ExecuteSkill.Parameter[2].Name := 'TargetPosition Z';
ExecuteSkill.Parameter[2].Value := 0 ;



ExecuteSkill.Parameter[4].ID := 4;
ExecuteSkill.Parameter[4].Name := 'Acceleration';
ExecuteSkill.Parameter[4].Value := 2000 ;


(*
ExecuteSkill.Parameter[5].ID := ;
ExecuteSkill.Parameter[5].Name := '';
ExecuteSkill.Parameter[5].Value := ;
*)



ExecuteSkill();

StepDone := ExecuteSkill.Done;
END_ACTION

ACTION Block2_active:
StepDone := FALSE;

//Skill auswählen
ExecuteSkill.SkillID 		:= 1315;
ExecuteSkill.SkillName	 	:= 'Block';

//Parameter setzen

ExecuteSkill.Parameter[1].ID := 1;
ExecuteSkill.Parameter[1].Name := 'TaskID';
ExecuteSkill.Parameter[1].Value := 130;


(*
ExecuteSkill.Parameter[2].ID := ;
ExecuteSkill.Parameter[2].Name := '';
ExecuteSkill.Parameter[2].Value := ;
*)

(*
ExecuteSkill.Parameter[3].ID := ;
ExecuteSkill.Parameter[3].Name := '';
ExecuteSkill.Parameter[3].Value := ;
*)

(*
ExecuteSkill.Parameter[4].ID := ;
ExecuteSkill.Parameter[4].Name := '';
ExecuteSkill.Parameter[4].Value := ;
*)

(*
ExecuteSkill.Parameter[5].ID := ;
ExecuteSkill.Parameter[5].Name := '';
ExecuteSkill.Parameter[5].Value := ;
*)



ExecuteSkill();

StepDone := ExecuteSkill.Done;
END_ACTION

ACTION Reserve_active:
StepDone := FALSE;
RecipeDone := FALSE;
//Skill auswählen
ExecuteSkill.SkillID 		:= 1310;
ExecuteSkill.SkillName	 	:= 'Reserve';

//Parameter setzen

ExecuteSkill.Parameter[1].ID := 1;
ExecuteSkill.Parameter[1].Name := 'TaskID';
ExecuteSkill.Parameter[1].Value := 123;


(*
ExecuteSkill.Parameter[2].ID := ;
ExecuteSkill.Parameter[2].Name := '';
ExecuteSkill.Parameter[2].Value := ;
*)

(*
ExecuteSkill.Parameter[3].ID := ;
ExecuteSkill.Parameter[3].Name := '';
ExecuteSkill.Parameter[3].Value := ;
*)

(*
ExecuteSkill.Parameter[4].ID := ;
ExecuteSkill.Parameter[4].Name := '';
ExecuteSkill.Parameter[4].Value := ;
*)

(*
ExecuteSkill.Parameter[5].ID := ;
ExecuteSkill.Parameter[5].Name := '';
ExecuteSkill.Parameter[5].Value := ;
*)



ExecuteSkill();

StepDone := ExecuteSkill.Done;
END_ACTION

ACTION Unblock_active:
StepDone := FALSE;

//Skill auswählen
ExecuteSkill.SkillID 		:= 1316;
ExecuteSkill.SkillName	 	:= 'Unblock';

//Parameter setzen

ExecuteSkill.Parameter[1].ID := 1;
ExecuteSkill.Parameter[1].Name := 'TaskID';
ExecuteSkill.Parameter[1].Value := 125;


(*
ExecuteSkill.Parameter[2].ID := ;
ExecuteSkill.Parameter[2].Name := '';
ExecuteSkill.Parameter[2].Value := ;
*)

(*
ExecuteSkill.Parameter[3].ID := ;
ExecuteSkill.Parameter[3].Name := '';
ExecuteSkill.Parameter[3].Value := ;
*)

(*
ExecuteSkill.Parameter[4].ID := ;
ExecuteSkill.Parameter[4].Name := '';
ExecuteSkill.Parameter[4].Value := ;
*)

(*
ExecuteSkill.Parameter[5].ID := ;
ExecuteSkill.Parameter[5].Name := '';
ExecuteSkill.Parameter[5].Value := ;
*)



ExecuteSkill();

StepDone := ExecuteSkill.Done;
END_ACTION

ACTION Cookie_active:
StepDone := FALSE;
RecipeDone := FALSE;
//Skill auswählen
ExecuteSkill.SkillID 		:= 1010;
ExecuteSkill.SkillName	 	:= 'Cookie ausgeben';





ExecuteSkill();

StepDone := ExecuteSkill.Done;
END_ACTION

ACTION TransOutput_active:
StepDone := FALSE;

//Skill auswählen
ExecuteSkill.SkillID 		:= 1320;
ExecuteSkill.SkillName	 	:= 'Name';

//Parameter setzen

ExecuteSkill.Parameter[3].ID := 3;
ExecuteSkill.Parameter[3].Name := 'Velocity';
ExecuteSkill.Parameter[3].Value := 1500;



ExecuteSkill.Parameter[4].ID := 4 ;
ExecuteSkill.Parameter[4].Name := 'Acceleration';
ExecuteSkill.Parameter[4].Value := 1000 ;



ExecuteSkill.Parameter[1].ID := 1;
ExecuteSkill.Parameter[1].Name := 'TargetPosition X';
ExecuteSkill.Parameter[1].Value := 3200 ;
ExecuteSkill.Parameter[1].StringValue := '#DP#2#XPosition' ;




ExecuteSkill.Parameter[2].ID := 2;
ExecuteSkill.Parameter[2].Name := 'TargetPosition Z';
ExecuteSkill.Parameter[2].Value := ZInputOutput;


(*
ExecuteSkill.Parameter[5].ID := ;
ExecuteSkill.Parameter[5].Name := '';
ExecuteSkill.Parameter[5].Value := ;
*)



ExecuteSkill();

StepDone := ExecuteSkill.Done;
END_ACTION

ACTION TransportToTopping_active:
StepDone := FALSE;

//Skill auswählen
ExecuteSkill.SkillID 		:= 1320;
ExecuteSkill.SkillName	 	:= 'Transport';

//Parameter setzen

ExecuteSkill.Parameter[3].ID := 3;
ExecuteSkill.Parameter[3].Name := 'Velocity';
ExecuteSkill.Parameter[3].Value := 1000;



ExecuteSkill.Parameter[1].ID :=  1;
ExecuteSkill.Parameter[1].Name := 'TargetPosition X';
ExecuteSkill.Parameter[1].Value := 30 ;
ExecuteSkill.Parameter[1].StringValue := '#DP#2#XPosition';



ExecuteSkill.Parameter[2].ID := 2;
ExecuteSkill.Parameter[2].Name := 'TargetPosition Z';
ExecuteSkill.Parameter[2].Value := ZCremeModule + ZCremeModuleCalibration - Layercnt * ( cookiethickness + toppingthickness);

ExecuteSkill();

StepDone := ExecuteSkill.Done;
END_ACTION

ACTION Unblock_active_0:
StepDone := FALSE;

//Skill auswählen
ExecuteSkill.SkillID 		:= 1316;
ExecuteSkill.SkillName	 	:= 'Unblock';

//Parameter setzen

ExecuteSkill.Parameter[1].ID := 1;
ExecuteSkill.Parameter[1].Name := 'TaskID';
ExecuteSkill.Parameter[1].Value := 128 ;


(*
ExecuteSkill.Parameter[2].ID := ;
ExecuteSkill.Parameter[2].Name := '';
ExecuteSkill.Parameter[2].Value := ;
*)

(*
ExecuteSkill.Parameter[3].ID := ;
ExecuteSkill.Parameter[3].Name := '';
ExecuteSkill.Parameter[3].Value := ;
*)

(*
ExecuteSkill.Parameter[4].ID := ;
ExecuteSkill.Parameter[4].Name := '';
ExecuteSkill.Parameter[4].Value := ;
*)

(*
ExecuteSkill.Parameter[5].ID := ;
ExecuteSkill.Parameter[5].Name := '';
ExecuteSkill.Parameter[5].Value := ;
*)



ExecuteSkill();

StepDone := ExecuteSkill.Done;
END_ACTION

ACTION Cookie_exit:
Layercnt := Layercnt +1;
END_ACTION

ACTION Block0_active:
StepDone := FALSE;

//Skill auswählen

CASE LREAL_TO_INT (order.UserParameter[2].Value) OF

1:
ExecuteSkill.SkillID 		:= 1315;
ExecuteSkill.SkillName	 	:= 'Block';

ExecuteSkill();

StepDone := ExecuteSkill.Done;
ELSE StepDone := TRUE;

END_CASE
END_ACTION

ACTION BlockBeiTopping_active:
StepDone := FALSE;

//Skill auswählen
ExecuteSkill.SkillID 		:= 1315;
ExecuteSkill.SkillName	 	:= 'Block';

//Parameter setzen

ExecuteSkill.Parameter[1].ID := 1;
ExecuteSkill.Parameter[1].Name := 'TaskID';
ExecuteSkill.Parameter[1].Value := 130;


(*
ExecuteSkill.Parameter[2].ID := ;
ExecuteSkill.Parameter[2].Name := '';
ExecuteSkill.Parameter[2].Value := ;
*)

(*
ExecuteSkill.Parameter[3].ID := ;
ExecuteSkill.Parameter[3].Name := '';
ExecuteSkill.Parameter[3].Value := ;
*)

(*
ExecuteSkill.Parameter[4].ID := ;
ExecuteSkill.Parameter[4].Name := '';
ExecuteSkill.Parameter[4].Value := ;
*)

(*
ExecuteSkill.Parameter[5].ID := ;
ExecuteSkill.Parameter[5].Name := '';
ExecuteSkill.Parameter[5].Value := ;
*)



ExecuteSkill();

StepDone := ExecuteSkill.Done;
END_ACTION

ACTION Completed_active:
RecipeDone := TRUE;
StepDone := FALSE;
Layercnt := 0;
END_ACTION

ACTION ErsterKeks_active:
StepDone := FALSE;
RecipeDone := FALSE;
//Skill auswählen
ExecuteSkill.SkillID 		:= 1010;
ExecuteSkill.SkillName	 	:= 'Seperate Cookie';


ExecuteSkill();

StepDone := ExecuteSkill.Done;
END_ACTION

ACTION Output_active:
StepDone := FALSE;

//Skill auswählen
ExecuteSkill.SkillID 		:= 1403;
ExecuteSkill.SkillName	 	:= 'Output';

//Parameter setzen

ExecuteSkill.Parameter[1].ID := 1;
ExecuteSkill.Parameter[1].Name := 'TaskID';
ExecuteSkill.Parameter[1].Value := Order.TaskID;


(*
ExecuteSkill.Parameter[2].ID := ;
ExecuteSkill.Parameter[2].Name := '';
ExecuteSkill.Parameter[2].Value := ;
*)

(*
ExecuteSkill.Parameter[3].ID := ;
ExecuteSkill.Parameter[3].Name := '';
ExecuteSkill.Parameter[3].Value := ;
*)

(*
ExecuteSkill.Parameter[4].ID := ;
ExecuteSkill.Parameter[4].Name := '';
ExecuteSkill.Parameter[4].Value := ;
*)

(*
ExecuteSkill.Parameter[5].ID := ;
ExecuteSkill.Parameter[5].Name := '';
ExecuteSkill.Parameter[5].Value := ;
*)



ExecuteSkill();

StepDone := ExecuteSkill.Done;
END_ACTION

ACTION Block1_active:
StepDone := FALSE;

//Skill auswählen
ExecuteSkill.SkillID 		:= 1315;
ExecuteSkill.SkillName	 	:= 'Block';

//Parameter setzen

ExecuteSkill.Parameter[1].ID := 1;
ExecuteSkill.Parameter[1].Name := 'TaskID';
ExecuteSkill.Parameter[1].Value := 127;


(*
ExecuteSkill.Parameter[2].ID := ;
ExecuteSkill.Parameter[2].Name := '';
ExecuteSkill.Parameter[2].Value := ;
*)

(*
ExecuteSkill.Parameter[3].ID := ;
ExecuteSkill.Parameter[3].Name := '';
ExecuteSkill.Parameter[3].Value := ;
*)

(*
ExecuteSkill.Parameter[4].ID := ;
ExecuteSkill.Parameter[4].Name := '';
ExecuteSkill.Parameter[4].Value := ;
*)

(*
ExecuteSkill.Parameter[5].ID := ;
ExecuteSkill.Parameter[5].Name := '';
ExecuteSkill.Parameter[5].Value := ;
*)



ExecuteSkill();

StepDone := ExecuteSkill.Done;
END_ACTION

ACTION Init_active:
RecipeDone := FALSE;

// Initialisation of Recipe Parameters an name etc
RecipeInfo.Name := 'Triple Cookie';
RecipeInfo.Description := 'Three Butter Cookies framing your choosen Toppings';
RecipeInfo.Dummy := FALSE;
RecipeInfo.RecipeID := 10018;	// 
Initdone := TRUE;
FOR i := 0 TO UserParameterCnt DO
	IF Order.UserParameter[i].Value = 0 THEN
		order.UserParameter[i].Value := RecipeInfo.UserParameter[i].Default;
	END_IF
END_FOR

//Parameter 0:

	RecipeInfo.UserParameter[0].Dummy 		:= FALSE;
	RecipeInfo.UserParameter[0].Default		:= 1;
	RecipeInfo.UserParameter[0].Description	:= 'Choose your first Topping (Top Layer)';
	RecipeInfo.UserParameter[0].MaxValue	:= 2;
	RecipeInfo.UserParameter[0].MinValue	:= 1;
	RecipeInfo.UserParameter[0].Name		:= 'Topping';
	RecipeInfo.UserParameter[0].Unit		:= 'Strawberry, Apple';
	RecipeInfo.UserParameter[0].Step		:= 1;

//Parameter 1:

	RecipeInfo.UserParameter[1].Dummy 		:= FALSE;
	RecipeInfo.UserParameter[1].Default		:= 50;
	RecipeInfo.UserParameter[1].Description	:= 'Amount of the selected Topping';
	RecipeInfo.UserParameter[1].MaxValue	:= 100;
	RecipeInfo.UserParameter[1].MinValue	:= 0;
	RecipeInfo.UserParameter[1].Name		:= 'Amount';
	RecipeInfo.UserParameter[1].Unit		:= '';
	RecipeInfo.UserParameter[1].Step		:= 1;

//Parameter 2:
	RecipeInfo.UserParameter[2].Dummy 		:= FALSE;
	RecipeInfo.UserParameter[2].Default		:= 2;
	RecipeInfo.UserParameter[2].Description	:= 'Choose weather you want to include a simulated module';
	RecipeInfo.UserParameter[2].MaxValue	:= 2;
	RecipeInfo.UserParameter[2].MinValue	:= 1;
	RecipeInfo.UserParameter[2].Name		:= 'Virtual Module';
	RecipeInfo.UserParameter[2].Unit		:= 'enabled, disabled';
	RecipeInfo.UserParameter[2].Step		:= 1;

//Parameter 3:
	RecipeInfo.UserParameter[3].Dummy 		:= FALSE;
	RecipeInfo.UserParameter[3].Default		:= 1;
	RecipeInfo.UserParameter[3].Description	:= 'Amount of the selected Topping';
	RecipeInfo.UserParameter[3].MaxValue	:= 100;
	RecipeInfo.UserParameter[3].MinValue	:= 0;
	RecipeInfo.UserParameter[3].Name		:= 'Amount';
	RecipeInfo.UserParameter[3].Unit		:= '';
	RecipeInfo.UserParameter[3].Step		:= 1;
//Parameter 4:

	RecipeInfo.UserParameter[4].Dummy 		:= FALSE;
	RecipeInfo.UserParameter[4].Default		:= 1;
	RecipeInfo.UserParameter[4].Description	:= 'Choose your third Topping';
	RecipeInfo.UserParameter[4].MaxValue	:= 2;
	RecipeInfo.UserParameter[4].MinValue	:= 1;
	RecipeInfo.UserParameter[4].Name		:= 'Topping';
	RecipeInfo.UserParameter[4].Unit		:= 'Strawberry, Apple';
	RecipeInfo.UserParameter[4].Step		:= 1;
	(*
//Parameter 5:

	RecipeInfo.UserParameter[5].Dummy 		:= FALSE;
	RecipeInfo.UserParameter[5].Default		:= 50;
	RecipeInfo.UserParameter[5].Description	:= 'Amount of the selected Topping';
	RecipeInfo.UserParameter[5].MaxValue	:= 100;
	RecipeInfo.UserParameter[5].MinValue	:= 0;
	RecipeInfo.UserParameter[5].Name		:= 'Amount';
	RecipeInfo.UserParameter[5].Unit		:= '';
	RecipeInfo.UserParameter[5].Step		:= 1;
*)
END_ACTION

ACTION Unblock3_active:
StepDone := FALSE;

//Skill auswählen
ExecuteSkill.SkillID 		:= 1316;
ExecuteSkill.SkillName	 	:= 'Unblock';

//Parameter setzen

ExecuteSkill.Parameter[1].ID := 1;
ExecuteSkill.Parameter[1].Name := 'TaskID';
ExecuteSkill.Parameter[1].Value := 131;


(*
ExecuteSkill.Parameter[2].ID := ;
ExecuteSkill.Parameter[2].Name := '';
ExecuteSkill.Parameter[2].Value := ;
*)

(*
ExecuteSkill.Parameter[3].ID := ;
ExecuteSkill.Parameter[3].Name := '';
ExecuteSkill.Parameter[3].Value := ;
*)

(*
ExecuteSkill.Parameter[4].ID := ;
ExecuteSkill.Parameter[4].Name := '';
ExecuteSkill.Parameter[4].Value := ;
*)

(*
ExecuteSkill.Parameter[5].ID := ;
ExecuteSkill.Parameter[5].Name := '';
ExecuteSkill.Parameter[5].Value := ;
*)



ExecuteSkill();

StepDone := ExecuteSkill.Done;
END_ACTION

ACTION Production0_active:
StepDone := FALSE;
RecipeDone := FALSE; 
//simulation ausgewählt?
CASE LREAL_TO_INT (order.UserParameter[2].Value) OF

1:
ExecuteSkill.SkillID 		:= 1337;
ExecuteSkill.SkillName	 	:= 'Testskill';

ExecuteSkill();

StepDone := ExecuteSkill.Done;
ELSE StepDone := TRUE;

END_CASE
END_ACTION

ACTION UnblockOutput_active:
StepDone := FALSE;

//Skill auswählen
ExecuteSkill.SkillID 		:= 1316;
ExecuteSkill.SkillName	 	:= 'Unblock';

//Parameter setzen



(*
ExecuteSkill.Parameter[2].ID := ;
ExecuteSkill.Parameter[2].Name := '';
ExecuteSkill.Parameter[2].Value := ;
*)

(*
ExecuteSkill.Parameter[3].ID := ;
ExecuteSkill.Parameter[3].Name := '';
ExecuteSkill.Parameter[3].Value := ;
*)

(*
ExecuteSkill.Parameter[4].ID := ;
ExecuteSkill.Parameter[4].Name := '';
ExecuteSkill.Parameter[4].Value := ;
*)

(*
ExecuteSkill.Parameter[5].ID := ;
ExecuteSkill.Parameter[5].Name := '';
ExecuteSkill.Parameter[5].Value := ;
*)



ExecuteSkill();

StepDone := ExecuteSkill.Done;
END_ACTION

ACTION Transport1_active:
StepDone := FALSE;

//Skill auswählen
ExecuteSkill.SkillID 		:= 1320;
ExecuteSkill.SkillName	 	:= 'Transport';

//Parameter setzen

ExecuteSkill.Parameter[3].ID := 3;
ExecuteSkill.Parameter[3].Name := 'Velocity';
ExecuteSkill.Parameter[3].Value := 1500;



ExecuteSkill.Parameter[4].ID := 4 ;
ExecuteSkill.Parameter[4].Name := 'Acceleration';
ExecuteSkill.Parameter[4].Value := 1000 ;



ExecuteSkill.Parameter[1].ID := 1;
ExecuteSkill.Parameter[1].Name := 'TargetPosition X';
ExecuteSkill.Parameter[1].Value := 3200 ;
ExecuteSkill.Parameter[1].StringValue := '#DP#2#XPosition' ;




ExecuteSkill.Parameter[2].ID := 2;
ExecuteSkill.Parameter[2].Name := 'TargetPosition Z';
ExecuteSkill.Parameter[2].Value := ZCookieModule + ZCocktailModuleCalibration;


(*
ExecuteSkill.Parameter[5].ID := ;
ExecuteSkill.Parameter[5].Name := '';
ExecuteSkill.Parameter[5].Value := ;
*)



ExecuteSkill();

StepDone := ExecuteSkill.Done;
END_ACTION

ACTION Unreserve_active:
StepDone := FALSE;

//Skill auswählen
ExecuteSkill.SkillID 		:= 1311;
ExecuteSkill.SkillName	 	:= 'Unreserve';

//Parameter setzen

ExecuteSkill.Parameter[1].ID := 1;
ExecuteSkill.Parameter[1].Name := 'TaskID';
ExecuteSkill.Parameter[1].Value := 131;


(*
ExecuteSkill.Parameter[2].ID := ;
ExecuteSkill.Parameter[2].Name := '';
ExecuteSkill.Parameter[2].Value := ;
*)

(*
ExecuteSkill.Parameter[3].ID := ;
ExecuteSkill.Parameter[3].Name := '';
ExecuteSkill.Parameter[3].Value := ;
*)

(*
ExecuteSkill.Parameter[4].ID := ;
ExecuteSkill.Parameter[4].Name := '';
ExecuteSkill.Parameter[4].Value := ;
*)

(*
ExecuteSkill.Parameter[5].ID := ;
ExecuteSkill.Parameter[5].Name := '';
ExecuteSkill.Parameter[5].Value := ;
*)



ExecuteSkill();

StepDone := ExecuteSkill.Done;
END_ACTION

ACTION Unblock2_active:
StepDone := FALSE;

//Skill auswählen
ExecuteSkill.SkillID 		:= 1316;
ExecuteSkill.SkillName	 	:= 'Unblock';

//Parameter setzen

ExecuteSkill.Parameter[1].ID := 1;
ExecuteSkill.Parameter[1].Name := 'TaskID';
ExecuteSkill.Parameter[1].Value := 131;


(*
ExecuteSkill.Parameter[2].ID := ;
ExecuteSkill.Parameter[2].Name := '';
ExecuteSkill.Parameter[2].Value := ;
*)

(*
ExecuteSkill.Parameter[3].ID := ;
ExecuteSkill.Parameter[3].Name := '';
ExecuteSkill.Parameter[3].Value := ;
*)

(*
ExecuteSkill.Parameter[4].ID := ;
ExecuteSkill.Parameter[4].Name := '';
ExecuteSkill.Parameter[4].Value := ;
*)

(*
ExecuteSkill.Parameter[5].ID := ;
ExecuteSkill.Parameter[5].Name := '';
ExecuteSkill.Parameter[5].Value := ;
*)



ExecuteSkill();

StepDone := ExecuteSkill.Done;
END_ACTION

ACTION unblock1_active_0:
StepDone := FALSE;

//Skill auswählen
ExecuteSkill.SkillID 		:= 1316;
ExecuteSkill.SkillName	 	:= 'Unblock';

//Parameter setzen

ExecuteSkill.Parameter[1].ID := 1;
ExecuteSkill.Parameter[1].Name := 'TaskID';
ExecuteSkill.Parameter[1].Value := 128 ;


(*
ExecuteSkill.Parameter[2].ID := ;
ExecuteSkill.Parameter[2].Name := '';
ExecuteSkill.Parameter[2].Value := ;
*)

(*
ExecuteSkill.Parameter[3].ID := ;
ExecuteSkill.Parameter[3].Name := '';
ExecuteSkill.Parameter[3].Value := ;
*)

(*
ExecuteSkill.Parameter[4].ID := ;
ExecuteSkill.Parameter[4].Name := '';
ExecuteSkill.Parameter[4].Value := ;
*)

(*
ExecuteSkill.Parameter[5].ID := ;
ExecuteSkill.Parameter[5].Name := '';
ExecuteSkill.Parameter[5].Value := ;
*)



ExecuteSkill();

StepDone := ExecuteSkill.Done;
END_ACTION

ACTION Transport3_active:
StepDone := FALSE;

//Skill auswählen
ExecuteSkill.SkillID 		:= 1320;
ExecuteSkill.SkillName	 	:= 'Transport';

//Parameter setzen

ExecuteSkill.Parameter[3].ID := 3;
ExecuteSkill.Parameter[3].Name := 'Velocity';
ExecuteSkill.Parameter[3].Value := 2800;



ExecuteSkill.Parameter[1].ID :=  1;
ExecuteSkill.Parameter[1].Name := 'TargetPosition X';
ExecuteSkill.Parameter[1].Value := 30 ;
ExecuteSkill.Parameter[1].StringValue := '#DP#-2#XPosition';



ExecuteSkill.Parameter[2].ID := 2;
ExecuteSkill.Parameter[2].Name := 'TargetPosition Z';
ExecuteSkill.Parameter[2].Value := 90;// ZCookieModule - ZCookieModuleCalibration - 2* Cookiethickness + toppingthickness+ Preasureheight  ;



ExecuteSkill.Parameter[4].ID := 4;
ExecuteSkill.Parameter[4].Name := 'Acceleration';
ExecuteSkill.Parameter[4].Value := 2000 ;


(*
ExecuteSkill.Parameter[5].ID := ;
ExecuteSkill.Parameter[5].Name := '';
ExecuteSkill.Parameter[5].Value := ;
*)



ExecuteSkill();

StepDone := ExecuteSkill.Done;
END_ACTION

END_FUNCTION_BLOCK

// ---- POUs/Recipes/Recipe_10030_HandModule.TcPOU
FUNCTION_BLOCK Recipe_10030_HandModule
VAR_INPUT
	execute	: BOOL;
	Order	: DUT_RECIPEORDER;
END_VAR
VAR_OUTPUT
	RecipeInfo	: DUT_RECIPEOFFER;
	RecipeDone	: BOOL;	
	InitDone	: BOOL;
END_VAR
VAR
	StepDone	: BOOL;
END_VAR

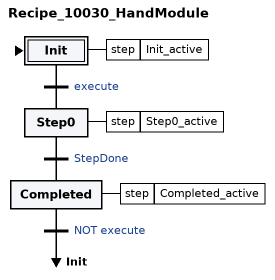
INITIAL_STEP Init:
    Init_active(N);  // step action
END_STEP
TRANSITION FROM Init TO Step0
    := execute;
END_TRANSITION
STEP Step0:
    Step0_active(N);  // step action
END_STEP
TRANSITION FROM Step0 TO Completed
    := StepDone;
END_TRANSITION
STEP Completed:
    Completed_active(N);  // step action
END_STEP
TRANSITION FROM Completed TO Init
    := NOT execute;
END_TRANSITION

ACTION Step6_active:
StepDone := FALSE;

//Skill auswählen
ExecuteSkill.SkillID 		:= 0000;
ExecuteSkill.SkillName	 	:= 'Name';

//Parameter setzen
(*
ExecuteSkill.Parameter[1].ID := 3;
ExecuteSkill.Parameter[1].Name := 'Velocity';
ExecuteSkill.Parameter[1].Value := 3000;
*)

(*
ExecuteSkill.Parameter[2].ID := ;
ExecuteSkill.Parameter[2].Name := '';
ExecuteSkill.Parameter[2].Value := ;
*)

(*
ExecuteSkill.Parameter[3].ID := ;
ExecuteSkill.Parameter[3].Name := '';
ExecuteSkill.Parameter[3].Value := ;
*)

(*
ExecuteSkill.Parameter[4].ID := ;
ExecuteSkill.Parameter[4].Name := '';
ExecuteSkill.Parameter[4].Value := ;
*)

(*
ExecuteSkill.Parameter[5].ID := ;
ExecuteSkill.Parameter[5].Name := '';
ExecuteSkill.Parameter[5].Value := ;
*)



ExecuteSkill();

StepDone := ExecuteSkill.Done;
END_ACTION

ACTION Step4_active:
StepDone := FALSE;

//Skill auswählen
ExecuteSkill.SkillID 		:= 0000;
ExecuteSkill.SkillName	 	:= 'Name';

//Parameter setzen
(*
ExecuteSkill.Parameter[1].ID := 3;
ExecuteSkill.Parameter[1].Name := 'Velocity';
ExecuteSkill.Parameter[1].Value := 3000;
*)

(*
ExecuteSkill.Parameter[2].ID := ;
ExecuteSkill.Parameter[2].Name := '';
ExecuteSkill.Parameter[2].Value := ;
*)

(*
ExecuteSkill.Parameter[3].ID := ;
ExecuteSkill.Parameter[3].Name := '';
ExecuteSkill.Parameter[3].Value := ;
*)

(*
ExecuteSkill.Parameter[4].ID := ;
ExecuteSkill.Parameter[4].Name := '';
ExecuteSkill.Parameter[4].Value := ;
*)

(*
ExecuteSkill.Parameter[5].ID := ;
ExecuteSkill.Parameter[5].Name := '';
ExecuteSkill.Parameter[5].Value := ;
*)



ExecuteSkill();

StepDone := ExecuteSkill.Done;
END_ACTION

ACTION Step2_active:
StepDone := FALSE;

//Skill auswählen
ExecuteSkill.SkillID 		:= 0000;
ExecuteSkill.SkillName	 	:= 'Name';

//Parameter setzen
(*
ExecuteSkill.Parameter[1].ID := 3;
ExecuteSkill.Parameter[1].Name := 'Velocity';
ExecuteSkill.Parameter[1].Value := 3000;
*)

(*
ExecuteSkill.Parameter[2].ID := ;
ExecuteSkill.Parameter[2].Name := '';
ExecuteSkill.Parameter[2].Value := ;
*)

(*
ExecuteSkill.Parameter[3].ID := ;
ExecuteSkill.Parameter[3].Name := '';
ExecuteSkill.Parameter[3].Value := ;
*)

(*
ExecuteSkill.Parameter[4].ID := ;
ExecuteSkill.Parameter[4].Name := '';
ExecuteSkill.Parameter[4].Value := ;
*)

(*
ExecuteSkill.Parameter[5].ID := ;
ExecuteSkill.Parameter[5].Name := '';
ExecuteSkill.Parameter[5].Value := ;
*)



ExecuteSkill();

StepDone := ExecuteSkill.Done;
END_ACTION

ACTION Step8_active:
StepDone := FALSE;

//Skill auswählen
ExecuteSkill.SkillID 		:= 0000;
ExecuteSkill.SkillName	 	:= 'Name';

//Parameter setzen
(*
ExecuteSkill.Parameter[1].ID := 3;
ExecuteSkill.Parameter[1].Name := 'Velocity';
ExecuteSkill.Parameter[1].Value := 3000;
*)

(*
ExecuteSkill.Parameter[2].ID := ;
ExecuteSkill.Parameter[2].Name := '';
ExecuteSkill.Parameter[2].Value := ;
*)

(*
ExecuteSkill.Parameter[3].ID := ;
ExecuteSkill.Parameter[3].Name := '';
ExecuteSkill.Parameter[3].Value := ;
*)

(*
ExecuteSkill.Parameter[4].ID := ;
ExecuteSkill.Parameter[4].Name := '';
ExecuteSkill.Parameter[4].Value := ;
*)

(*
ExecuteSkill.Parameter[5].ID := ;
ExecuteSkill.Parameter[5].Name := '';
ExecuteSkill.Parameter[5].Value := ;
*)



ExecuteSkill();

StepDone := ExecuteSkill.Done;
END_ACTION

ACTION Init_active:
RecipeDone := FALSE;

// Initialisation of Recipe Parameters an name etc
RecipeInfo.Name := 'Sample Product Name';
RecipeInfo.Description := 'This Recipe produces a product, which is very productive';
RecipeInfo.Dummy := FALSE;
RecipeInfo.RecipeID := 10000; 	// 
Initdone := TRUE;

//Parameter 1:
(*
	RecipeInfo.UserParameter[1].Dummy 		:= 
	RecipeInfo.UserParameter[1].Default		:=
	RecipeInfo.UserParameter[1].Description	:=
	RecipeInfo.UserParameter[1].MaxValue	:=
	RecipeInfo.UserParameter[1].MinValue	:=
	RecipeInfo.UserParameter[1].Name		:=
	RecipeInfo.UserParameter[1].Unit		:=
*)
//Parameter 2:

(*
	RecipeInfo.UserParameter[2].Dummy 		:= 
	RecipeInfo.UserParameter[2].Default		:=
	RecipeInfo.UserParameter[2].Description	:=
	RecipeInfo.UserParameter[2].MaxValue	:=
	RecipeInfo.UserParameter[2].MinValue	:=
	RecipeInfo.UserParameter[2].Name		:=
	RecipeInfo.UserParameter[2].Unit		:=
*)

//Parameter 3:

(*
	RecipeInfo.UserParameter[3].Dummy 		:= 
	RecipeInfo.UserParameter[3].Default		:=
	RecipeInfo.UserParameter[3].Description	:=
	RecipeInfo.UserParameter[3].MaxValue	:=
	RecipeInfo.UserParameter[3].MinValue	:=
	RecipeInfo.UserParameter[3].Name		:=
	RecipeInfo.UserParameter[3].Unit		:=
*)

//Parameter 4:

(*
	RecipeInfo.UserParameter[4].Dummy 		:= 
	RecipeInfo.UserParameter[4].Default		:=
	RecipeInfo.UserParameter[4].Description	:=
	RecipeInfo.UserParameter[4].MaxValue	:=
	RecipeInfo.UserParameter[4].MinValue	:=
	RecipeInfo.UserParameter[4].Name		:=
	RecipeInfo.UserParameter[4].Unit		:=
*)


//Parameter 5:

(*
	RecipeInfo.UserParameter[5].Dummy 		:= 
	RecipeInfo.UserParameter[5].Default		:=
	RecipeInfo.UserParameter[5].Description	:=
	RecipeInfo.UserParameter[5].MaxValue	:=
	RecipeInfo.UserParameter[5].MinValue	:=
	RecipeInfo.UserParameter[5].Name		:=
	RecipeInfo.UserParameter[5].Unit		:=
*)
END_ACTION

ACTION Step10_active:
StepDone := FALSE;

